		IF PULSO_CNT_L4_1T.Q = FALSE AND PULSO_CNT_L4_2T.Q = FALSE AND PULSO_CNT_L4_3T.Q = FALSE  THEN
		HabTemParadaL4 := TRUE;
		
		ELSE 	
		HabTemParadaL4 := FALSE;
		END_IF
		//LÓGICA PARA CONTAR TEMPO DE PARADA
//==============Habilita contadores 1º turno ================
IF (hora = HoraInicio1Turno AND minuto = MinInicio1Turno)  THEN
HabContL4_1T := TRUE;
HabContL4_3T := FALSE;
HabContL4_2T := FALSE;
CNT_PRD_L4_3T := 0;
CNT_PRD_L4_2T := 0;
CNT_PRD_L4_1T := 0;
TempoProduzindoL4 :=0;
EficL4_1T_projetada:=0;
EficL4_1T_realtime :=0;
ProdL4_1T_realtime :=0;
TempoParadaL4 :=0;
CXS_ATRASOL4:=0;
END_IF 


//==============Contador e Eficiencia L4 1 TURNO de cartuchos==========
IF HabContL4_1T = TRUE THEN 
PULSO_CNT_L4_1T(CLK:=CNT_L4);
//TMR_SIMUL_CNT1(IN:=LIBERA_TMR_SIMUL ,PT:=T#9S);	
		IF PULSO_CNT_L4_1T.Q = TRUE THEN
		CNT_PRD_L4_1T := CNT_PRD_L4_1T+1;
		//LIBERA_TMR_SIMUL := FALSE;
		RegistraHora := FALSE;
		MinDispTurnoAtual := MinDispL4_1T;
//ELSE 	
	//LIBERA_TMR_SIMUL:= TRUE;
		END_IF
		
			IF hora > 5 AND hora < 11 THEN

		ProdL4_1T_realtime := (INT_TO_REAL(ProducaoProgramada_L4_1T) / (MinDispL4_1T)) * ((
		(INT_TO_REAL(hora)-INT_TO_REAL(HoraInicio1Turno))*60)-INT_TO_REAL(MinInicio1Turno) + INT_TO_REAL(minuto));
		
		TempoProduzindoL4 :=  ((hora-HoraInicio1Turno)*60)-MinInicio1Turno+ minuto-TempoParadaL4;
		
		EficL4_1T_realtime := ( INT_TO_REAL(CNT_PRD_L4_1T) / ProdL4_1T_realtime ) * 100 * (EficL4_1T_projetada/100);
		EficL4_1T_projetada := (ProdL4_1T_realtime / ProducaoProgramada_L4_1T) * 100;
		END_IF
		
			IF hora > 11 AND hora < 15 THEN

		ProdL4_1T_realtime := (INT_TO_REAL(ProducaoProgramada_L4_1T) / (MinDispL4_1T)) * ((
		(INT_TO_REAL(hora)-INT_TO_REAL(HoraInicio1Turno))*60)-INT_TO_REAL(MinInicio1Turno) + INT_TO_REAL(minuto)-10-60);
		
		TempoProduzindoL4 :=  ((hora-HoraInicio1Turno)*60)-MinInicio1Turno+ minuto-TempoParadaL4;
		
		EficL4_1T_realtime := ( INT_TO_REAL(CNT_PRD_L4_1T) / ProdL4_1T_realtime ) * 100 * (EficL4_1T_projetada/100);
		EficL4_1T_projetada := (ProdL4_1T_realtime / ProducaoProgramada_L4_1T) * 100;
		END_IF
	
END_IF
EficienciaL4_1T := (INT_TO_REAL(CNT_PRD_L4_1T) / INT_TO_REAL(ProducaoProgramada_L4_1T) ) * 100;


//=====================1º TURNO ========================

//=====================2º TURNO ========================

	//10 minutos - Reunião / DSS / Treinamento
	//20 minutosPartida de linha / Parada de Linha
	//15 minutosRefeições (Café / Almoço / Janta)
	//60 minutosRefeições (Café / Almoço / Janta)
	//10 minutosPartida de linha / Parada de Linha
	IF hora = 0 THEN 
		hora := 24;
	END_IF
	
		MinDispL4_2T := (((INT_TO_REAL (HoraFim2Turno) - INT_TO_REAL(HoraInicio2Turno) )*60)-
		INT_TO_REAL(MinInicio2Turno)+INT_TO_REAL(MinFim2Turno)-60-10);
	
//==============Contador e Eficiencia L4 2 TURNO de cartuchos==========
//==============Habilita contadores 2º turno ================
IF (hora = HoraInicio2Turno AND minuto = MinInicio2Turno)  THEN
HabContL4_2T := TRUE;
HabContL4_1T := FALSE;
CNT_PRD_L4_3T := 0;
CNT_PRD_L4_2T := 0;
CNT_PRD_L4_1T := 0;
TempoParadaL4 :=0;
TempoProduzindoL4 :=0;
EficL4_1T_projetada:=0;
EficL4_1T_realtime :=0;
ProdL4_1T_realtime :=0;
TempoParadaL4 :=0;
CXS_ATRASOL4:=0;
END_IF 
IF HabContL4_2T = TRUE THEN 
PULSO_CNT_L4_2T(CLK:=CNT_L4);
//TMR_SIMUL_CNT2(IN:=LIBERA_TMR_SIMUL4T ,PT:=T#7S);
		IF PULSO_CNT_L4_2T.Q = TRUE  THEN
		CNT_PRD_L4_2T := CNT_PRD_L4_2T+1;
		//LIBERA_TMR_SIMUL4T := FALSE;
		MinDispTurnoAtual := MinDispL4_2T;
//ELSE 	
	//LIBERA_TMR_SIMUL4T:= TRUE;	
		END_IF
		CNT_PRD_L4_1T := CNT_PRD_L4_2T ;
		EficL4_1T_projetada:=EficL4_2T_projetada;
		EficL4_1T_realtime :=EficL4_2T_realtime;
		ProdL4_1T_realtime :=ProdL4_1T_realtime;
		
			IF hora > 13 AND hora < 19 THEN

		ProdL4_2T_realtime := (INT_TO_REAL(ProducaoProgramada_L4_T2) / (MinDispL4_2T)) * ((
		(INT_TO_REAL(hora)-INT_TO_REAL(HoraInicio2Turno))*60)-INT_TO_REAL(MinInicio2Turno) + INT_TO_REAL(minuto));
		
		TempoProduzindoL4 :=  ((hora-HoraInicio2Turno)*60)-MinInicio2Turno+ minuto-TempoParadaL4;
		
		EficL4_2T_realtime := ( INT_TO_REAL(CNT_PRD_L4_2T) / ProdL4_2T_realtime ) * 100 * (EficL4_2T_projetada/100);
		EficL4_2T_projetada := (ProdL4_2T_realtime / ProducaoProgramada_L4_T2) * 100;
		END_IF
		IF hora > 19 AND hora < 23 THEN

		ProdL4_2T_realtime := (INT_TO_REAL(ProducaoProgramada_L4_T2) / (MinDispL4_2T)) * ((
		(INT_TO_REAL(hora)-INT_TO_REAL(HoraInicio2Turno))*60)-INT_TO_REAL(MinInicio2Turno) + INT_TO_REAL(minuto)-10-60);
		
		TempoProduzindoL4 :=  ((hora-HoraInicio2Turno)*60)-MinInicio2Turno+ minuto-TempoParadaL4;
		
		EficL4_2T_realtime := ( INT_TO_REAL(CNT_PRD_L4_2T) / ProdL4_2T_realtime ) * 100 * (EficL4_2T_projetada/100);
		EficL4_2T_projetada := (ProdL4_2T_realtime / ProducaoProgramada_L4_T2) * 100;
		END_IF
END_IF
EficienciaL4_2T := (INT_TO_REAL (CNT_PRD_L4_2T) / INT_TO_REAL (ProducaoProgramada_L4_T2)  ) * 100;

//=====================2º TURNO ========================

//=====================3º TURNO ========================
//==============Contador e Eficiencia L4 3 TURNO de cartuchos==========

//==============Habilita contadores 3º turno ================
//10 minutos - Reunião / DSS / Treinamento
	//20 minutosPartida de linha / Parada de Linha
	//15 minutosRefeições (Café / Almoço / Janta)
	//60 minutosRefeições (Café / Almoço / Janta)
	//10 minutosPartida de linha / Parada de Linha
	IF hora = 0 THEN 
		hora := 24;
	END_IF
	
		MinDispL4_3T := (((INT_TO_REAL (HoraFim3Turno) - INT_TO_REAL(HoraInicio3Turno) )*60)-
		INT_TO_REAL(MinInicio3Turno)+INT_TO_REAL(MinFim3Turno)-60-10);
		
	
//==============Contador e Eficiencia L4 3 TURNO de cartuchos==========
//==============Habilita contadores 3º turno ================
IF (hora = HoraInicio3Turno AND minuto = MinInicio3Turno)  THEN
HabContL4_3T := TRUE;
HabContL4_2T := FALSE;
HabContL4_1T := FALSE;
CNT_PRD_L4_3T := 0;
CNT_PRD_L4_2T := 0;
CNT_PRD_L4_1T := 0;
TempoParadaL4 :=0;
TempoProduzindoL4 :=0;
EficL4_1T_projetada:=0;
EficL4_1T_realtime :=0;
ProdL4_1T_realtime :=0;
TempoParadaL4 :=0;
CXS_ATRASOL4:=0;
END_IF 

IF HabContL4_3T = TRUE THEN 
PULSO_CNT_L4_3T(CLK:=CNT_L4);	
		IF PULSO_CNT_L4_3T.Q = TRUE THEN
		CNT_PRD_L4_3T := CNT_PRD_L4_3T+1;	
			CNT_PRD_L4_1T := CNT_PRD_L4_3T ;
		EficL4_1T_projetada:=EficL4_3T_projetada;
		EficL4_1T_realtime :=EficL4_3T_realtime;
		ProdL4_1T_realtime :=ProdL4_3T_realtime;
		END_IF
		IF hora > 21 AND hora <= 24 THEN

		ProdL4_3T_realtime := (INT_TO_REAL(ProducaoProgramada_L4_T3) / (MinDispL4_3T)) * ((
		(INT_TO_REAL(hora)-INT_TO_REAL(HoraInicio3Turno))*60)-INT_TO_REAL(MinInicio3Turno) + INT_TO_REAL(minuto));
		
		TempoProduzindoL4 :=  ((hora-HoraInicio3Turno)*60)-MinInicio3Turno+ minuto-TempoParadaL4;
	
		EficL4_3T_realtime := ( INT_TO_REAL(CNT_PRD_L4_3T) / ProdL4_3T_realtime ) * 100 *(EficL4_3T_projetada/100) ;
		EficL4_3T_projetada := (ProdL4_3T_realtime / ProducaoProgramada_L4_T3) * 100;
		END_IF
		IF ((hora > 0 ) AND minuto > 30) AND hora < 2 THEN

		ProdL4_3T_realtime := (INT_TO_REAL(ProducaoProgramada_L4_T3) / (MinDispL4_3T)) * ((
		(INT_TO_REAL(hora)-INT_TO_REAL(HoraInicio3Turno))*60)-INT_TO_REAL(MinInicio3Turno) + INT_TO_REAL(minuto)-10-60);
		
		TempoProduzindoL4 :=  ((hora-HoraInicio3Turno)*60)-MinInicio3Turno+ minuto-TempoParadaL4;
	
		EficL4_3T_realtime := ( INT_TO_REAL(CNT_PRD_L4_3T) / ProdL4_3T_realtime ) * 100 *(EficL4_3T_projetada/100) ;
		EficL4_3T_projetada := (ProdL4_3T_realtime / ProducaoProgramada_L4_T3) * 100;
		END_IF
END_IF


EficienciaL4_3T := (INT_TO_REAL (CNT_PRD_L4_3T) / INT_TO_REAL (ProducaoProgramada_L4_T3)  ) * 100;


IF (hora = HoraInicio3Turno AND minuto = MinInicio3Turno)  THEN
HabContL4_3T := TRUE;
HabContL4_2T := FALSE;
END_IF 

IF HabContL4_3T = TRUE THEN 
PULSO_CNT_L4_3T(CLK:=CNT_L4);
//TMR_SIMUL_CNT3(IN:=LIBERA_TMR_SIMUL4T ,PT:=T#8S);
		IF PULSO_CNT_L4_3T.Q = TRUE  THEN
		CNT_PRD_L4_3T := CNT_PRD_L4_3T+1;
		//LIBERA_TMR_SIMUL4T := FALSE;
		MinDispTurnoAtual := MinDispL4_3T;
//ELSE 	
	//LIBERA_TMR_SIMUL4T:= TRUE;	
		END_IF
		END_IF
	
	
EficienciaL4_3T := (INT_TO_REAL (CNT_PRD_L4_3T) / INT_TO_REAL(ProducaoProgramada_L4_T3)  ) * 100;
//=====================3º TURNO ========================

IF (hora = 11 AND minuto = 0) OR (hora = 19 AND minuto = 0) OR (hora = 1 AND minuto = 30)  THEN
	refeicao := TRUE;
	END_IF
	IF (hora = 11 AND minuto = 40) OR  (hora = 20 AND minuto = 0)  OR  (hora = 2 AND minuto = 30)  THEN
	refeicao := FALSE;
	END_IF 
	
	IF (hora = 6 AND minuto = 0) OR (hora = 20 AND minuto = 0) OR (hora = 2 AND minuto = 30)  THEN
	DDS := TRUE;
	END_IF
	IF (hora = 6 AND minuto = 10) OR  (hora = 20 AND minuto = 10)  OR  (hora = 2 AND minuto = 40)  THEN
	DDS := FALSE;
	END_IF 
	IF (hora = 6 AND minuto = 0) OR (hora = 14 AND minuto = 20) OR (hora = 22 AND minuto = 30)  THEN
	SETUP := TRUE;
	END_IF
	IF (hora = 6 AND minuto = 30) OR  (hora = 14 AND minuto = 50)  OR  (hora = 23 AND minuto = 0)  THEN
	SETUP := FALSE;
	END_IF 
	
	
//STATUS DA LINHA 4
//STATUS DO EQUIPAMENTO
//0- SEM PROGRAMAÇÃO
//1- PRODUZINDO
//2- PARADA
//3- REFEIÇÃO
//4- DDS
//5- SETUP

	
IF ProducaoProgramada_L4_1T = 0 AND HabContL4_1T  AND TempParadaL4.Q = TRUE THEN
	Status_L4 := 0;
	L4semprogramacao :=TRUE;
	END_IF
		IF ProducaoProgramada_L4_1T > 0 AND HabContL4_1T = TRUE THEN 
		L4semprogramacao :=FALSE;
		END_IF
	
IF ProducaoProgramada_L4_T2 = 0 AND HabContL4_2T = TRUE AND TempParadaL4.Q = TRUE THEN
	Status_L4 := 0;
	L4semprogramacao :=TRUE;
		END_IF
			IF ProducaoProgramada_L4_T2 > 0 AND HabContL4_2T = TRUE THEN 
				L4semprogramacao :=FALSE;
				END_IF
				
IF ProducaoProgramada_L4_T3 = 0 AND HabContL4_3T = TRUE AND TempParadaL4.Q = TRUE THEN
	Status_L4 := 0;
	L4semprogramacao :=TRUE;
		END_IF
			IF ProducaoProgramada_L4_T3 > 0 AND HabContL4_3T = TRUE THEN 
			L4semprogramacao :=FALSE;
			END_IF
	
IF  TempParadaL4.Q = FALSE  THEN
	Status_L4 := 1;
END_IF

	IF refeicao = FALSE AND SETUP = FALSE AND DDS = FALSE AND TempParadaL4.Q = TRUE AND L4semprogramacao = FALSE THEN
	Status_L4 := 2;
	END_IF

IF refeicao = TRUE AND TempParadaL4.Q = TRUE  THEN
Status_L4 := 3;
END_IF

IF DDS = TRUE AND TempParadaL4.Q = TRUE THEN
Status_L4 := 4;
END_IF

//IF SETUP = TRUE THEN
//Status_L4 := 5;
//END_IF
//STATUS DA LINHA 4

END_PROGRAM

// Device/Application/ProdL5
PROGRAM ProdL5
VAR
	//PRODUÇÃO LINHAS ENVASE
	
//=========================	
PULSO_CNT_L5_1T: R_TRIG;
PULSO_CNT_L5_2T: R_TRIG;
PULSO_CNT_L5_3T: R_TRIG;
	CNT_PRD_L5: INT;
	//CNT_L5: BOOL;
//=========================	
	Result : RTC_STATUS;
	DATEANDTIME : EXTENDED_DATE_AND_TIME;
	xEnable : BOOL;
//=========================		
	dia: INT;
	mes: INT;
	ano: INT;
	hora: INT;
	minuto: INT;
	segundo: INT;
	
	
	
	//HoraInicio1Turno: INT;
	//MinInicio1Turno: INT;
	HoraFim1Turno: INT;
	MinFim1Turno: INT;
	//HoraInicio2Turno: INT;
	//MinInicio2Turno: INT;
	HoraFim2Turno: INT;
	MinFim2Turno: INT;
	//HoraInicio3Turno: INT;
	//MinInicio3Turno: INT;
	HoraFim3Turno: INT;
	MinFim3Turno: INT;
	EficienciaL5: INT;
	
	
	HabContL5_1T: BOOL;
	HabContL5_2T: BOOL;
	HabContL5_3T: BOOL;
	
	CNT_PRD_L5_2T: INT;
	CNT_PRD_L5_3T: INT;
	EficienciaL5_1T: REAL;
	EficienciaL5_2T: REAL;
	EficienciaL5_3T: REAL;
	
	MinDispL5_1T: REAL;
	
	ProdL5_1T_realtime: REAL;
	MinDispL5_2T: REAL;
	ProdL5_2T_realtime: REAL;
	EficL5_2T_realtime: REAL;
	MinDispL5_3T: REAL;
	ProdL5_3T_realtime: REAL;
	EficL5_3T_realtime: REAL;
	
	//TMR_SIMUL_CNT1: TON;
	//LIBERA_TMR_SIMUL: BOOL;
	EficL5_2T_projetada: REAL;
	//TMR_SIMUL_CNT2: TON;
	//LIBERA_TMR_SIMUL5T: BOOL;
	//TMR_SIMUL_CNT3: TON;
	//LIBERA_TMR_SIMUL5T: BOOL;
	EficL5_3T_projetada: REAL;
//	EficL5_1T_realtime: REAL;
	HabTemParadaL5: BOOL;
	TempParadaL5: Ton;
	horaParadaL5: INT;
	MinParadaL5: INT;
	RegistraHora: BOOL;
	Borda_des_RegistraHora: F_TRIG;
	HoraRetornoParadaL5: INT;
	MinRetornoParadaL5: INT;
	TempoParadaL5L5: INT;
	TotalMinParado: TON;
	HabTotalMinParado: BOOL;
	//TempoProduzindoL5: REAL;
	//MinDispTurnoAtual: REAL;

	refeicao: BOOL;
	DDS: BOOL;
	SETUP: BOOL;
	L5semprogramacao: BOOL;
END_VAR


//LÓGICA PARA ANÁLISES DE PRODUTIVADADE DA L5 DE CARTUCHOS
	dia := BYTE_TO_INT (DATEANDTIME.byDayOfMonth);
	mes := BYTE_TO_INT (DATEANDTIME.byMonth);
	ano := WORD_TO_INT (DATEANDTIME.wYear);
	hora := BYTE_TO_INT (DATEANDTIME.byHours);
	minuto := BYTE_TO_INT (DATEANDTIME.byMinutes);
	segundo := BYTE_TO_INT (DATEANDTIME.bySeconds);
	xEnable := TRUE;
	
	//HABILITA RTC==========================
	IF xEnable = TRUE THEN
	Result := GetDateAndTime(DATEANDTIME);
	END_IF
//HABILITA RTC==========================

//=====================1º TURNO ========================
	
		//HoraInicio1Turno: INT;
	
	HoraFim1Turno:= HoraInicio2Turno;
	MinFim1Turno:= MinInicio2Turno;
	HoraFim2Turno:= HoraInicio3Turno;
	MinFim2Turno:= MinInicio3Turno;
	
	//10 minutos - Reunião / DSS / Treinamento
	//20 minutosPartida de linha / Parada de Linha xxxxxxxxxx
	//15 minutosRefeições (Café / Almoço / Janta)xxxxxxxxxxxx
	//60 minutosRefeições (Café / Almoço / Janta)
	//10 minutosPartida de linha / Parada de Linha xxxxxxxxxxxxxx
			
	MinDispL5_1T := (((INT_TO_REAL (HoraFim1Turno) - INT_TO_REAL(HoraInicio1Turno) )*60)-
		INT_TO_REAL(MinInicio1Turno)+INT_TO_REAL(MinFim1Turno)-60-10);
		
			IF TempoProduzindoL5 < 1 THEN
			TempoProduzindoL5 :=0;
		END_IF
	
			//LÓGICA PARA VERIFICAR SE EXISTE ATRASO DE PRODUÇÃO NO INSTANTE ATUAL
		
	IF  CXS_ATRASOL5 >= 0 AND HabContL5_1T = TRUE THEN 
	CXS_ATRASOL5:= REAL_TO_INT(ProdL5_1T_realtime)-CNT_PRD_L5_1T;
	END_IF
	IF  CXS_ATRASOL5 >= 0 AND HabContL5_2T = TRUE THEN 
	CXS_ATRASOL5:= REAL_TO_INT(ProdL5_2T_realtime)-CNT_PRD_L5_1T;
	END_IF
	IF  CXS_ATRASOL5 >= 0 AND HabContL5_3T = TRUE THEN 
	CXS_ATRASOL5:=REAL_TO_INT(ProdL5_2T_realtime)-CNT_PRD_L5_1T;
	END_IF
		IF  CXS_ATRASOL5  < 0 THEN 
		CXS_ATRASOL5:= 0;
		END_IF
	
	
	//LÓGICA PARA VERIFICAR SE EXISTE ATRASO DE PRODUÇÃO NO INSTANTE ATUAL
	
		
		//LÓGICA PARA CONTAR TEMPO DE PARADA
		TempParadaL5(IN:=HabTemParadaL5 ,PT:= T#30S);
		IF TempParadaL5.Q   THEN
		TotalMinParado(IN:=HabTotalMinParado ,PT:= T#1M);
		IF TotalMinParado.Q = TRUE THEN
			TempoParadaL5 := TempoParadaL5+1;
			HabTotalMinParado := FALSE;
			ELSE
				HabTotalMinParado := TRUE;
			END_IF
		END_IF
		
		IF PULSO_CNT_L5_1T.Q = FALSE AND PULSO_CNT_L5_2T.Q = FALSE AND PULSO_CNT_L5_3T.Q = FALSE  THEN
		HabTemParadaL5 := TRUE;
		
		ELSE 	
		HabTemParadaL5 := FALSE;
		END_IF
		//LÓGICA PARA CONTAR TEMPO DE PARADA
//==============Habilita contadores 1º turno ================
IF (hora = HoraInicio1Turno AND minuto = MinInicio1Turno)  THEN
HabContL5_1T := TRUE;
HabContL5_3T := FALSE;
HabContL5_2T := FALSE;
CNT_PRD_L5_3T := 0;
CNT_PRD_L5_2T := 0;
CNT_PRD_L5_1T := 0;
TempoProduzindoL5 :=0;
EficL5_1T_projetada:=0;
EficL5_1T_realtime :=0;
ProdL5_1T_realtime :=0;
TempoParadaL5 :=0;
CXS_ATRASOL5:=0;
END_IF 


//==============Contador e Eficiencia L5 1 TURNO de cartuchos==========
IF HabContL5_1T = TRUE THEN 
PULSO_CNT_L5_1T(CLK:=CNT_L5);
//TMR_SIMUL_CNT1(IN:=LIBERA_TMR_SIMUL ,PT:=T#9S);	
		IF PULSO_CNT_L5_1T.Q = TRUE THEN
		CNT_PRD_L5_1T := CNT_PRD_L5_1T+1;
		//LIBERA_TMR_SIMUL := FALSE;
		RegistraHora := FALSE;
		MinDispTurnoAtual := MinDispL5_1T;
//ELSE 	
	//LIBERA_TMR_SIMUL:= TRUE;
		END_IF
		
			IF hora > 5 AND hora < 11 THEN

		ProdL5_1T_realtime := (INT_TO_REAL(ProducaoProgramada_L5_1T) / (MinDispL5_1T)) * ((
		(INT_TO_REAL(hora)-INT_TO_REAL(HoraInicio1Turno))*60)-INT_TO_REAL(MinInicio1Turno) + INT_TO_REAL(minuto));
		
		TempoProduzindoL5 :=  ((hora-HoraInicio1Turno)*60)-MinInicio1Turno+ minuto-TempoParadaL5;
		
		EficL5_1T_realtime := ( INT_TO_REAL(CNT_PRD_L5_1T) / ProdL5_1T_realtime ) * 100 * (EficL5_1T_projetada/100);
		EficL5_1T_projetada := (ProdL5_1T_realtime / ProducaoProgramada_L5_1T) * 100;
		END_IF
		
			IF hora > 11 AND hora < 15 THEN

		ProdL5_1T_realtime := (INT_TO_REAL(ProducaoProgramada_L5_1T) / (MinDispL5_1T)) * ((
		(INT_TO_REAL(hora)-INT_TO_REAL(HoraInicio1Turno))*60)-INT_TO_REAL(MinInicio1Turno) + INT_TO_REAL(minuto)-10-60);
		
		TempoProduzindoL5 :=  ((hora-HoraInicio1Turno)*60)-MinInicio1Turno+ minuto-TempoParadaL5;
		
		EficL5_1T_realtime := ( INT_TO_REAL(CNT_PRD_L5_1T) / ProdL5_1T_realtime ) * 100 * (EficL5_1T_projetada/100);
		EficL5_1T_projetada := (ProdL5_1T_realtime / ProducaoProgramada_L5_1T) * 100;
		END_IF
	
END_IF
EficienciaL5_1T := (INT_TO_REAL(CNT_PRD_L5_1T) / INT_TO_REAL(ProducaoProgramada_L5_1T) ) * 100;


//=====================1º TURNO ========================

//=====================2º TURNO ========================

	//10 minutos - Reunião / DSS / Treinamento
	//20 minutosPartida de linha / Parada de Linha
	//15 minutosRefeições (Café / Almoço / Janta)
	//60 minutosRefeições (Café / Almoço / Janta)
	//10 minutosPartida de linha / Parada de Linha
	IF hora = 0 THEN 
		hora := 24;
	END_IF
	
		MinDispL5_2T := (((INT_TO_REAL (HoraFim2Turno) - INT_TO_REAL(HoraInicio2Turno) )*60)-
		INT_TO_REAL(MinInicio2Turno)+INT_TO_REAL(MinFim2Turno)-60-10);
	
//==============Contador e Eficiencia L5 2 TURNO de cartuchos==========
//==============Habilita contadores 2º turno ================
IF (hora = HoraInicio2Turno AND minuto = MinInicio2Turno)  THEN
HabContL5_2T := TRUE;
HabContL5_1T := FALSE;
CNT_PRD_L5_3T := 0;
CNT_PRD_L5_2T := 0;
CNT_PRD_L5_1T := 0;
TempoParadaL5 :=0;
TempoProduzindoL5 :=0;
EficL5_1T_projetada:=0;
EficL5_1T_realtime :=0;
ProdL5_1T_realtime :=0;
TempoParadaL5 :=0;
CXS_ATRASOL5:=0;
END_IF 
IF HabContL5_2T = TRUE THEN 
PULSO_CNT_L5_2T(CLK:=CNT_L5);
//TMR_SIMUL_CNT2(IN:=LIBERA_TMR_SIMUL5T ,PT:=T#7S);
		IF PULSO_CNT_L5_2T.Q = TRUE  THEN
		CNT_PRD_L5_2T := CNT_PRD_L5_2T+1;
		//LIBERA_TMR_SIMUL5T := FALSE;
		MinDispTurnoAtual := MinDispL5_2T;
//ELSE 	
	//LIBERA_TMR_SIMUL5T:= TRUE;	
		END_IF
		CNT_PRD_L5_1T := CNT_PRD_L5_2T ;
		EficL5_1T_projetada:=EficL5_2T_projetada;
		EficL5_1T_realtime :=EficL5_2T_realtime;
		ProdL5_1T_realtime :=ProdL5_1T_realtime;
		
			IF hora > 13 AND hora < 19 THEN

		ProdL5_2T_realtime := (INT_TO_REAL(ProducaoProgramada_L5_T2) / (MinDispL5_2T)) * ((
		(INT_TO_REAL(hora)-INT_TO_REAL(HoraInicio2Turno))*60)-INT_TO_REAL(MinInicio2Turno) + INT_TO_REAL(minuto));
		
		TempoProduzindoL5 :=  ((hora-HoraInicio2Turno)*60)-MinInicio2Turno+ minuto-TempoParadaL5;
		
		EficL5_2T_realtime := ( INT_TO_REAL(CNT_PRD_L5_2T) / ProdL5_2T_realtime ) * 100 * (EficL5_2T_projetada/100);
		EficL5_2T_projetada := (ProdL5_2T_realtime / ProducaoProgramada_L5_T2) * 100;
		END_IF
		IF hora > 19 AND hora < 23 THEN

		ProdL5_2T_realtime := (INT_TO_REAL(ProducaoProgramada_L5_T2) / (MinDispL5_2T)) * ((
		(INT_TO_REAL(hora)-INT_TO_REAL(HoraInicio2Turno))*60)-INT_TO_REAL(MinInicio2Turno) + INT_TO_REAL(minuto)-10-60);
		
		TempoProduzindoL5 :=  ((hora-HoraInicio2Turno)*60)-MinInicio2Turno+ minuto-TempoParadaL5;
		
		EficL5_2T_realtime := ( INT_TO_REAL(CNT_PRD_L5_2T) / ProdL5_2T_realtime ) * 100 * (EficL5_2T_projetada/100);
		EficL5_2T_projetada := (ProdL5_2T_realtime / ProducaoProgramada_L5_T2) * 100;
		END_IF
END_IF
EficienciaL5_2T := (INT_TO_REAL (CNT_PRD_L5_2T) / INT_TO_REAL (ProducaoProgramada_L5_T2)  ) * 100;

//=====================2º TURNO ========================

//=====================3º TURNO ========================
//==============Contador e Eficiencia L5 3 TURNO de cartuchos==========

//==============Habilita contadores 3º turno ================
//10 minutos - Reunião / DSS / Treinamento
	//20 minutosPartida de linha / Parada de Linha
	//15 minutosRefeições (Café / Almoço / Janta)
	//60 minutosRefeições (Café / Almoço / Janta)
	//10 minutosPartida de linha / Parada de Linha
	IF hora = 0 THEN 
		hora := 24;
	END_IF
	
		MinDispL5_3T := (((INT_TO_REAL (HoraFim3Turno) - INT_TO_REAL(HoraInicio3Turno) )*60)-
		INT_TO_REAL(MinInicio3Turno)+INT_TO_REAL(MinFim3Turno)-60-10);
		
	
//==============Contador e Eficiencia L5 3 TURNO de cartuchos==========
//==============Habilita contadores 3º turno ================
IF (hora = HoraInicio3Turno AND minuto = MinInicio3Turno)  THEN
HabContL5_3T := TRUE;
HabContL5_2T := FALSE;
HabContL5_1T := FALSE;
CNT_PRD_L5_3T := 0;
CNT_PRD_L5_2T := 0;
CNT_PRD_L5_1T := 0;
TempoParadaL5 :=0;
TempoProduzindoL5 :=0;
EficL5_1T_projetada:=0;
EficL5_1T_realtime :=0;
ProdL5_1T_realtime :=0;
TempoParadaL5 :=0;
CXS_ATRASOL5:=0;
END_IF 

IF HabContL5_3T = TRUE THEN 
PULSO_CNT_L5_3T(CLK:=CNT_L5);	
		IF PULSO_CNT_L5_3T.Q = TRUE THEN
		CNT_PRD_L5_3T := CNT_PRD_L5_3T+1;	
			CNT_PRD_L5_1T := CNT_PRD_L5_3T ;
		EficL5_1T_projetada:=EficL5_3T_projetada;
		EficL5_1T_realtime :=EficL5_3T_realtime;
		ProdL5_1T_realtime :=ProdL5_3T_realtime;
		END_IF
		IF hora > 21 AND hora <= 24 THEN

		ProdL5_3T_realtime := (INT_TO_REAL(ProducaoProgramada_L5_T3) / (MinDispL5_3T)) * ((
		(INT_TO_REAL(hora)-INT_TO_REAL(HoraInicio3Turno))*60)-INT_TO_REAL(MinInicio3Turno) + INT_TO_REAL(minuto));
		
		TempoProduzindoL5 :=  ((hora-HoraInicio3Turno)*60)-MinInicio3Turno+ minuto-TempoParadaL5;
	
		EficL5_3T_realtime := ( INT_TO_REAL(CNT_PRD_L5_3T) / ProdL5_3T_realtime ) * 100 *(EficL5_3T_projetada/100) ;
		EficL5_3T_projetada := (ProdL5_3T_realtime / ProducaoProgramada_L5_T3) * 100;
		END_IF
		IF ((hora > 0 ) AND minuto > 30) AND hora < 2 THEN

		ProdL5_3T_realtime := (INT_TO_REAL(ProducaoProgramada_L5_T3) / (MinDispL5_3T)) * ((
		(INT_TO_REAL(hora)-INT_TO_REAL(HoraInicio3Turno))*60)-INT_TO_REAL(MinInicio3Turno) + INT_TO_REAL(minuto)-10-60);
		
		TempoProduzindoL5 :=  ((hora-HoraInicio3Turno)*60)-MinInicio3Turno+ minuto-TempoParadaL5;
	
		EficL5_3T_realtime := ( INT_TO_REAL(CNT_PRD_L5_3T) / ProdL5_3T_realtime ) * 100 *(EficL5_3T_projetada/100) ;
		EficL5_3T_projetada := (ProdL5_3T_realtime / ProducaoProgramada_L5_T3) * 100;
		END_IF
END_IF


EficienciaL5_3T := (INT_TO_REAL (CNT_PRD_L5_3T) / INT_TO_REAL (ProducaoProgramada_L5_T3)  ) * 100;


IF (hora = HoraInicio3Turno AND minuto = MinInicio3Turno)  THEN
HabContL5_3T := TRUE;
HabContL5_2T := FALSE;
END_IF 

IF HabContL5_3T = TRUE THEN 
PULSO_CNT_L5_3T(CLK:=CNT_L5);
//TMR_SIMUL_CNT3(IN:=LIBERA_TMR_SIMUL5T ,PT:=T#8S);
		IF PULSO_CNT_L5_3T.Q = TRUE  THEN
		CNT_PRD_L5_3T := CNT_PRD_L5_3T+1;
		//LIBERA_TMR_SIMUL5T := FALSE;
		MinDispTurnoAtual := MinDispL5_3T;
//ELSE 	
	//LIBERA_TMR_SIMUL5T:= TRUE;	
		END_IF
		END_IF
	
	
EficienciaL5_3T := (INT_TO_REAL (CNT_PRD_L5_3T) / INT_TO_REAL(ProducaoProgramada_L5_T3)  ) * 100;
//=====================3º TURNO ========================

IF (hora = 11 AND minuto = 0) OR (hora = 19 AND minuto = 0) OR (hora = 1 AND minuto = 30)  THEN
	refeicao := TRUE;
	END_IF
	IF (hora = 11 AND minuto = 40) OR  (hora = 20 AND minuto = 0)  OR  (hora = 2 AND minuto = 30)  THEN
	refeicao := FALSE;
	END_IF 
	
	IF (hora = 6 AND minuto = 0) OR (hora = 20 AND minuto = 0) OR (hora = 2 AND minuto = 30)  THEN
	DDS := TRUE;
	END_IF
	IF (hora = 6 AND minuto = 10) OR  (hora = 20 AND minuto = 10)  OR  (hora = 2 AND minuto = 40)  THEN
	DDS := FALSE;
	END_IF 
	IF (hora = 6 AND minuto = 0) OR (hora = 14 AND minuto = 20) OR (hora = 22 AND minuto = 30)  THEN
	SETUP := TRUE;
	END_IF
	IF (hora = 6 AND minuto = 30) OR  (hora = 14 AND minuto = 50)  OR  (hora = 23 AND minuto = 0)  THEN
	SETUP := FALSE;
	END_IF 
	
//STATUS DA LINHA =5
//STATUS DO EQUIPAMENTO
//0- SEM PROGRAMAÇÃO
//1- PRODUZINDO
//2- PARADA
//3- REFEIÇÃO
//4- DDS
//5- SETUP

IF ProducaoProgramada_L5_1T = 0 AND HabContL5_1T = TRUE AND TempParadaL5.Q = TRUE THEN
	Status_L5 := 0;
	L5semprogramacao :=TRUE;
	END_IF
		IF ProducaoProgramada_L5_1T > 0 AND HabContL5_1T = TRUE THEN 
		L5semprogramacao :=FALSE;
		END_IF
	
IF ProducaoProgramada_L5_T2 = 0 AND HabContL5_2T = TRUE AND TempParadaL5.Q = TRUE THEN
	Status_L5 := 0;
	L5semprogramacao :=TRUE;
		END_IF
			IF ProducaoProgramada_L5_T2 > 0 AND HabContL5_2T = TRUE THEN 
				L5semprogramacao :=FALSE;
				END_IF
				
IF ProducaoProgramada_L5_T3 = 0 AND HabContL5_3T = TRUE AND TempParadaL5.Q = TRUE THEN
	Status_L5 := 0;
	L5semprogramacao :=TRUE;
		END_IF
			IF ProducaoProgramada_L5_T3 > 0 AND HabContL5_3T = TRUE THEN 
			L5semprogramacao :=FALSE;
			END_IF
	
IF  TempParadaL5.Q = FALSE  THEN
	Status_L5 := 1;
END_IF

	IF refeicao = FALSE AND SETUP = FALSE AND DDS = FALSE AND TempParadaL5.Q = TRUE AND L5semprogramacao = FALSE THEN
	Status_L5 := 2;
	END_IF

IF refeicao = TRUE  AND TempParadaL5.Q = TRUE THEN
Status_L5 := 3;
END_IF

IF DDS = TRUE  AND TempParadaL5.Q = TRUE THEN
Status_L5 := 4;
END_IF

//IF SETUP = TRUE THEN
//Status_L5 := 5;
//END_IF
//STATUS DA LINHA 5

END_PROGRAM

// Device/Application/ProdL6
PROGRAM ProdL6
VAR
	//PRODUÇÃO LINHAS ENVASE
	
//=========================	
PULSO_CNT_L6_1T: R_TRIG;
PULSO_CNT_L6_2T: R_TRIG;
PULSO_CNT_L6_3T: R_TRIG;
	CNT_PRD_L6: INT;
	//CNT_L6: BOOL;
//=========================	
	Result : RTC_STATUS;
	DATEANDTIME : EXTENDED_DATE_AND_TIME;
	xEnable : BOOL;
//=========================		
	dia: INT;
	mes: INT;
	ano: INT;
	hora: INT;
	minuto: INT;
	segundo: INT;
	
	
	
	//HoraInicio1Turno: INT;
	//MinInicio1Turno: INT;
	HoraFim1Turno: INT;
	MinFim1Turno: INT;
	//HoraInicio2Turno: INT;
	//MinInicio2Turno: INT;
	HoraFim2Turno: INT;
	MinFim2Turno: INT;
	//HoraInicio3Turno: INT;
	//MinInicio3Turno: INT;
	HoraFim3Turno: INT;
	MinFim3Turno: INT;
	EficienciaL6: INT;
	
	
	HabContL6_1T: BOOL;
	HabContL6_2T: BOOL;
	HabContL6_3T: BOOL;
	
	CNT_PRD_L6_2T: INT;
	CNT_PRD_L6_3T: INT;
	EficienciaL6_1T: REAL;
	EficienciaL6_2T: REAL;
	EficienciaL6_3T: REAL;
	
	MinDispL6_1T: REAL;
	
	ProdL6_1T_realtime: REAL;
	MinDispL6_2T: REAL;
	ProdL6_2T_realtime: REAL;
	EficL6_2T_realtime: REAL;
	MinDispL6_3T: REAL;
	ProdL6_3T_realtime: REAL;
	EficL6_3T_realtime: REAL;
	
	//TMR_SIMUL_CNT1: TON;
	//LIBERA_TMR_SIMUL: BOOL;
	EficL6_2T_projetada: REAL;
	//TMR_SIMUL_CNT2: TON;
	//LIBERA_TMR_SIMUL6T: BOOL;
	//TMR_SIMUL_CNT3: TON;
	//LIBERA_TMR_SIMUL3T: BOOL;
	EficL6_3T_projetada: REAL;
//	EficL6_1T_realtime: REAL;
	HabTemParadaL6: BOOL;
	TempParadaL6: Ton;
	horaParadaL6: INT;
	MinParadaL6: INT;
	RegistraHora: BOOL;
	Borda_des_RegistraHora: F_TRIG;
	HoraRetornoParadaL6: INT;
	MinRetornoParadaL6: INT;
	TempoParadaL6L6: INT;
	TotalMinParado: TON;
	HabTotalMinParado: BOOL;
	//TempoProduzindoL6: REAL;
	//MinDispTurnoAtual: REAL;

	refeicao: BOOL;
	DDS: BOOL;
	SETUP: BOOL;
	L6semprogramacao: BOOL;
END_VAR


//LÓGICA PARA ANÁLISES DE PRODUTIVADADE DA L6 DE CARTUCHOS
	dia := BYTE_TO_INT (DATEANDTIME.byDayOfMonth);
	mes := BYTE_TO_INT (DATEANDTIME.byMonth);
	ano := WORD_TO_INT (DATEANDTIME.wYear);
	hora := BYTE_TO_INT (DATEANDTIME.byHours);
	minuto := BYTE_TO_INT (DATEANDTIME.byMinutes);
	segundo := BYTE_TO_INT (DATEANDTIME.bySeconds);
	xEnable := TRUE;
	
	//HABILITA RTC==========================
	IF xEnable = TRUE THEN
	Result := GetDateAndTime(DATEANDTIME);
	END_IF
//HABILITA RTC==========================

//=====================1º TURNO ========================
	
		//HoraInicio1Turno: INT;
	
	HoraFim1Turno:= HoraInicio2Turno;
	MinFim1Turno:= MinInicio2Turno;
	HoraFim2Turno:= HoraInicio3Turno;
	MinFim2Turno:= MinInicio3Turno;
	
	//10 minutos - Reunião / DSS / Treinamento
	//20 minutosPartida de linha / Parada de Linha xxxxxxxxxx
	//15 minutosRefeições (Café / Almoço / Janta)xxxxxxxxxxxx
	//60 minutosRefeições (Café / Almoço / Janta)
	//10 minutosPartida de linha / Parada de Linha xxxxxxxxxxxxxx
			
	MinDispL6_1T := (((INT_TO_REAL (HoraFim1Turno) - INT_TO_REAL(HoraInicio1Turno) )*60)-
		INT_TO_REAL(MinInicio1Turno)+INT_TO_REAL(MinFim1Turno)-60-10);
		
		IF TempoProduzindoL6 < 1 THEN
			TempoProduzindoL6 :=0;
		END_IF
	
			//LÓGICA PARA VERIFICAR SE EXISTE ATRASO DE PRODUÇÃO NO INSTANTE ATUAL
		
	IF  CXS_ATRASOL6 >= 0 AND HabContL6_1T = TRUE THEN 
	CXS_ATRASOL6:= REAL_TO_INT(ProdL6_1T_realtime)-CNT_PRD_L6_1T;
	END_IF
	IF  CXS_ATRASOL6 >= 0 AND HabContL6_2T = TRUE THEN 
	CXS_ATRASOL6:= REAL_TO_INT(ProdL6_2T_realtime)-CNT_PRD_L6_1T;
	END_IF
	IF  CXS_ATRASOL6 >= 0 AND HabContL6_3T = TRUE THEN 
	CXS_ATRASOL6:=REAL_TO_INT(ProdL6_2T_realtime)-CNT_PRD_L6_1T;
	END_IF
		IF  CXS_ATRASOL6  < 0 THEN 
		CXS_ATRASOL6:= 0;
		END_IF
	
	//LÓGICA PARA VERIFICAR SE EXISTE ATRASO DE PRODUÇÃO NO INSTANTE ATUAL
		
		//LÓGICA PARA CONTAR TEMPO DE PARADA
		TempParadaL6(IN:=HabTemParadaL6 ,PT:= T#30S);
		IF TempParadaL6.Q   THEN
		TotalMinParado(IN:=HabTotalMinParado ,PT:= T#1M);
		IF TotalMinParado.Q = TRUE THEN
			TempoParadaL6 := TempoParadaL6+1;
			HabTotalMinParado := FALSE;
			ELSE
				HabTotalMinParado := TRUE;
			END_IF
		END_IF
		
		IF PULSO_CNT_L6_1T.Q = FALSE AND PULSO_CNT_L6_2T.Q = FALSE AND PULSO_CNT_L6_3T.Q = FALSE  THEN
		HabTemParadaL6 := TRUE;
		
		ELSE 	
		HabTemParadaL6 := FALSE;
		END_IF
		//LÓGICA PARA CONTAR TEMPO DE PARADA
//==============Habilita contadores 1º turno ================
IF (hora = HoraInicio1Turno AND minuto = MinInicio1Turno)  THEN
HabContL6_1T := TRUE;
HabContL6_3T := FALSE;
HabContL6_2T := FALSE;
CNT_PRD_L6_3T := 0;
CNT_PRD_L6_2T := 0;
CNT_PRD_L6_1T := 0;
TempoProduzindoL6 :=0;
EficL6_1T_projetada:=0;
EficL6_1T_realtime :=0;
ProdL6_1T_realtime :=0;
TempoParadaL6 :=0;
CXS_ATRASOL6:=0;
END_IF 


//==============Contador e Eficiencia L6 1 TURNO de cartuchos==========
IF HabContL6_1T = TRUE THEN 
PULSO_CNT_L6_1T(CLK:=CNT_L6);
//TMR_SIMUL_CNT1(IN:=LIBERA_TMR_SIMUL ,PT:=T#9S);	
		IF PULSO_CNT_L6_1T.Q = TRUE THEN
		CNT_PRD_L6_1T := CNT_PRD_L6_1T+1;
		//LIBERA_TMR_SIMUL := FALSE;
		RegistraHora := FALSE;
		MinDispTurnoAtual := MinDispL6_1T;
//ELSE 	
	//LIBERA_TMR_SIMUL:= TRUE;
		END_IF
		
			IF hora > 5 AND hora < 11 THEN

		ProdL6_1T_realtime := (INT_TO_REAL(ProducaoProgramada_L6_1T) / (MinDispL6_1T)) * ((
		(INT_TO_REAL(hora)-INT_TO_REAL(HoraInicio1Turno))*60)-INT_TO_REAL(MinInicio1Turno) + INT_TO_REAL(minuto));
		
		TempoProduzindoL6 :=  ((hora-HoraInicio1Turno)*60)-MinInicio1Turno+ minuto-TempoParadaL6;
		
		EficL6_1T_realtime := ( INT_TO_REAL(CNT_PRD_L6_1T) / ProdL6_1T_realtime ) * 100 * (EficL6_1T_projetada/100);
		EficL6_1T_projetada := (ProdL6_1T_realtime / ProducaoProgramada_L6_1T) * 100;
		END_IF
		
			IF hora > 11 AND hora < 15 THEN

		ProdL6_1T_realtime := (INT_TO_REAL(ProducaoProgramada_L6_1T) / (MinDispL6_1T)) * ((
		(INT_TO_REAL(hora)-INT_TO_REAL(HoraInicio1Turno))*60)-INT_TO_REAL(MinInicio1Turno) + INT_TO_REAL(minuto)-10-60);
		
		TempoProduzindoL6 :=  ((hora-HoraInicio1Turno)*60)-MinInicio1Turno+ minuto-TempoParadaL6;
		
		EficL6_1T_realtime := ( INT_TO_REAL(CNT_PRD_L6_1T) / ProdL6_1T_realtime ) * 100 * (EficL6_1T_projetada/100);
		EficL6_1T_projetada := (ProdL6_1T_realtime / ProducaoProgramada_L6_1T) * 100;
		END_IF
	
END_IF
EficienciaL6_1T := (INT_TO_REAL(CNT_PRD_L6_1T) / INT_TO_REAL(ProducaoProgramada_L6_1T) ) * 100;


//=====================1º TURNO ========================

//=====================2º TURNO ========================

	//10 minutos - Reunião / DSS / Treinamento
	//20 minutosPartida de linha / Parada de Linha
	//15 minutosRefeições (Café / Almoço / Janta)
	//60 minutosRefeições (Café / Almoço / Janta)
	//10 minutosPartida de linha / Parada de Linha
	IF hora = 0 THEN 
		hora := 24;
	END_IF
	
		MinDispL6_2T := (((INT_TO_REAL (HoraFim2Turno) - INT_TO_REAL(HoraInicio2Turno) )*60)-
		INT_TO_REAL(MinInicio2Turno)+INT_TO_REAL(MinFim2Turno)-60-10);
	
//==============Contador e Eficiencia L6 2 TURNO de cartuchos==========
//==============Habilita contadores 2º turno ================
IF (hora = HoraInicio2Turno AND minuto = MinInicio2Turno)  THEN
HabContL6_2T := TRUE;
HabContL6_1T := FALSE;
CNT_PRD_L6_3T := 0;
CNT_PRD_L6_2T := 0;
CNT_PRD_L6_1T := 0;
TempoParadaL6 :=0;
TempoProduzindoL6 :=0;
EficL6_1T_projetada:=0;
EficL6_1T_realtime :=0;
ProdL6_1T_realtime :=0;
TempoParadaL6 :=0;
CXS_ATRASOL6:=0;
END_IF 
IF HabContL6_2T = TRUE THEN 
PULSO_CNT_L6_2T(CLK:=CNT_L6);
//TMR_SIMUL_CNT2(IN:=LIBERA_TMR_SIMUL6T ,PT:=T#7S);
		IF PULSO_CNT_L6_2T.Q = TRUE  THEN
		CNT_PRD_L6_2T := CNT_PRD_L6_2T+1;
		//LIBERA_TMR_SIMUL6T := FALSE;
		MinDispTurnoAtual := MinDispL6_2T;
//ELSE 	
	//LIBERA_TMR_SIMUL6T:= TRUE;	
		END_IF
		CNT_PRD_L6_1T := CNT_PRD_L6_2T ;
		EficL6_1T_projetada:=EficL6_2T_projetada;
		EficL6_1T_realtime :=EficL6_2T_realtime;
		ProdL6_1T_realtime :=ProdL6_1T_realtime;
		
			IF hora > 13 AND hora < 19 THEN

		ProdL6_2T_realtime := (INT_TO_REAL(ProducaoProgramada_L6_T2) / (MinDispL6_2T)) * ((
		(INT_TO_REAL(hora)-INT_TO_REAL(HoraInicio2Turno))*60)-INT_TO_REAL(MinInicio2Turno) + INT_TO_REAL(minuto));
		
		TempoProduzindoL6 :=  ((hora-HoraInicio2Turno)*60)-MinInicio2Turno+ minuto-TempoParadaL6;
		
		EficL6_2T_realtime := ( INT_TO_REAL(CNT_PRD_L6_2T) / ProdL6_2T_realtime ) * 100 * (EficL6_2T_projetada/100);
		EficL6_2T_projetada := (ProdL6_2T_realtime / ProducaoProgramada_L6_T2) * 100;
		END_IF
		IF hora > 19 AND hora < 23 THEN

		ProdL6_2T_realtime := (INT_TO_REAL(ProducaoProgramada_L6_T2) / (MinDispL6_2T)) * ((
		(INT_TO_REAL(hora)-INT_TO_REAL(HoraInicio2Turno))*60)-INT_TO_REAL(MinInicio2Turno) + INT_TO_REAL(minuto)-10-60);
		
		TempoProduzindoL6 :=  ((hora-HoraInicio2Turno)*60)-MinInicio2Turno+ minuto-TempoParadaL6;
		
		EficL6_2T_realtime := ( INT_TO_REAL(CNT_PRD_L6_2T) / ProdL6_2T_realtime ) * 100 * (EficL6_2T_projetada/100);
		EficL6_2T_projetada := (ProdL6_2T_realtime / ProducaoProgramada_L6_T2) * 100;
		END_IF
END_IF
EficienciaL6_2T := (INT_TO_REAL (CNT_PRD_L6_2T) / INT_TO_REAL (ProducaoProgramada_L6_T2)  ) * 100;

//=====================2º TURNO ========================

//=====================3º TURNO ========================
//==============Contador e Eficiencia L6 3 TURNO de cartuchos==========

//==============Habilita contadores 3º turno ================
//10 minutos - Reunião / DSS / Treinamento
	//20 minutosPartida de linha / Parada de Linha
	//15 minutosRefeições (Café / Almoço / Janta)
	//60 minutosRefeições (Café / Almoço / Janta)
	//10 minutosPartida de linha / Parada de Linha
	IF hora = 0 THEN 
		hora := 24;
	END_IF
	
		MinDispL6_3T := (((INT_TO_REAL (HoraFim3Turno) - INT_TO_REAL(HoraInicio3Turno) )*60)-
		INT_TO_REAL(MinInicio3Turno)+INT_TO_REAL(MinFim3Turno)-60-10);
		
	
//==============Contador e Eficiencia L6 3 TURNO de cartuchos==========
//==============Habilita contadores 3º turno ================
IF (hora = HoraInicio3Turno AND minuto = MinInicio3Turno)  THEN
HabContL6_3T := TRUE;
HabContL6_2T := FALSE;
HabContL6_1T := FALSE;
CNT_PRD_L6_3T := 0;
CNT_PRD_L6_2T := 0;
CNT_PRD_L6_1T := 0;
TempoParadaL6 :=0;
TempoProduzindoL6 :=0;
EficL6_1T_projetada:=0;
EficL6_1T_realtime :=0;
ProdL6_1T_realtime :=0;
TempoParadaL6 :=0;
CXS_ATRASOL6:=0;
END_IF 

IF HabContL6_3T = TRUE THEN 
PULSO_CNT_L6_3T(CLK:=CNT_L6);	
		IF PULSO_CNT_L6_3T.Q = TRUE THEN
		CNT_PRD_L6_3T := CNT_PRD_L6_3T+1;	
			CNT_PRD_L6_1T := CNT_PRD_L6_3T ;
		EficL6_1T_projetada:=EficL6_3T_projetada;
		EficL6_1T_realtime :=EficL6_3T_realtime;
		ProdL6_1T_realtime :=ProdL6_3T_realtime;
		END_IF
		IF hora > 21 AND hora <= 24 THEN

		ProdL6_3T_realtime := (INT_TO_REAL(ProducaoProgramada_L6_T3) / (MinDispL6_3T)) * ((
		(INT_TO_REAL(hora)-INT_TO_REAL(HoraInicio3Turno))*60)-INT_TO_REAL(MinInicio3Turno) + INT_TO_REAL(minuto));
		
		TempoProduzindoL6 :=  ((hora-HoraInicio3Turno)*60)-MinInicio3Turno+ minuto-TempoParadaL6;
	
		EficL6_3T_realtime := ( INT_TO_REAL(CNT_PRD_L6_3T) / ProdL6_3T_realtime ) * 100 *(EficL6_3T_projetada/100) ;
		EficL6_3T_projetada := (ProdL6_3T_realtime / ProducaoProgramada_L6_T3) * 100;
		END_IF
		IF ((hora > 0 ) AND minuto > 30) AND hora < 2 THEN

		ProdL6_3T_realtime := (INT_TO_REAL(ProducaoProgramada_L6_T3) / (MinDispL6_3T)) * ((
		(INT_TO_REAL(hora)-INT_TO_REAL(HoraInicio3Turno))*60)-INT_TO_REAL(MinInicio3Turno) + INT_TO_REAL(minuto)-10-60);
		
		TempoProduzindoL6 :=  ((hora-HoraInicio3Turno)*60)-MinInicio3Turno+ minuto-TempoParadaL6;
	
		EficL6_3T_realtime := ( INT_TO_REAL(CNT_PRD_L6_3T) / ProdL6_3T_realtime ) * 100 *(EficL6_3T_projetada/100) ;
		EficL6_3T_projetada := (ProdL6_3T_realtime / ProducaoProgramada_L6_T3) * 100;
		END_IF
END_IF


EficienciaL6_3T := (INT_TO_REAL (CNT_PRD_L6_3T) / INT_TO_REAL (ProducaoProgramada_L6_T3)  ) * 100;


IF (hora = HoraInicio3Turno AND minuto = MinInicio3Turno)  THEN
HabContL6_3T := TRUE;
HabContL6_2T := FALSE;
END_IF 

IF HabContL6_3T = TRUE THEN 
PULSO_CNT_L6_3T(CLK:=CNT_L6);
//TMR_SIMUL_CNT3(IN:=LIBERA_TMR_SIMUL3T ,PT:=T#8S);
		IF PULSO_CNT_L6_3T.Q = TRUE  THEN
		CNT_PRD_L6_3T := CNT_PRD_L6_3T+1;
		//LIBERA_TMR_SIMUL3T := FALSE;
		MinDispTurnoAtual := MinDispL6_3T;
//ELSE 	
	//LIBERA_TMR_SIMUL3T:= TRUE;	
		END_IF
		END_IF
	
	
EficienciaL6_3T := (INT_TO_REAL (CNT_PRD_L6_3T) / INT_TO_REAL(ProducaoProgramada_L6_T3)  ) * 100;
//=====================3º TURNO ========================

IF (hora = 11 AND minuto = 0) OR (hora = 19 AND minuto = 0) OR (hora = 1 AND minuto = 30)  THEN
	refeicao := TRUE;
	END_IF
	IF (hora = 11 AND minuto = 40) OR  (hora = 20 AND minuto = 0)  OR  (hora = 2 AND minuto = 30)  THEN
	refeicao := FALSE;
	END_IF 
	
	IF (hora = 6 AND minuto = 0) OR (hora = 20 AND minuto = 0) OR (hora = 2 AND minuto = 30)  THEN
	DDS := TRUE;
	END_IF
	IF (hora = 6 AND minuto = 10) OR  (hora = 20 AND minuto = 10)  OR  (hora = 2 AND minuto = 40)  THEN
	DDS := FALSE;
	END_IF 
	IF (hora = 6 AND minuto = 0) OR (hora = 14 AND minuto = 20) OR (hora = 22 AND minuto = 30)  THEN
	SETUP := TRUE;
	END_IF
	IF (hora = 6 AND minuto = 30) OR  (hora = 14 AND minuto = 50)  OR  (hora = 23 AND minuto = 0)  THEN
	SETUP := FALSE;
	END_IF 

//STATUS DA LINHA 6
//STATUS DO EQUIPAMENTO
//0- SEM PROGRAMAÇÃO
//1- PRODUZINDO
//2- PARADA
//3- REFEIÇÃO
//4- DDS
//5- SETUP

IF ProducaoProgramada_L6_1T = 0 AND HabContL6_1T = TRUE AND TempParadaL6.Q = TRUE THEN
	Status_L6 := 0;
	L6semprogramacao :=TRUE;
	END_IF
		IF ProducaoProgramada_L6_1T > 0 AND HabContL6_1T = TRUE THEN 
		L6semprogramacao :=FALSE;
		END_IF
	
IF ProducaoProgramada_L6_T2 = 0 AND HabContL6_2T = TRUE AND TempParadaL6.Q = TRUE THEN
	Status_L6 := 0;
	L6semprogramacao :=TRUE;
		END_IF
			IF ProducaoProgramada_L6_T2 > 0 AND HabContL6_2T = TRUE THEN 
				L6semprogramacao :=FALSE;
				END_IF
				
IF ProducaoProgramada_L6_T3 = 0 AND HabContL6_3T = TRUE  AND TempParadaL6.Q = TRUE THEN
	Status_L6 := 0;
	L6semprogramacao :=TRUE;
		END_IF
			IF ProducaoProgramada_L6_T3 > 0 AND HabContL6_3T = TRUE THEN 
			L6semprogramacao :=FALSE;
			END_IF
	
IF TempParadaL6.Q = FALSE  THEN
	Status_L6 := 1;
END_IF

	IF refeicao = FALSE AND SETUP = FALSE AND DDS = FALSE AND TempParadaL6.Q = TRUE AND L6semprogramacao = FALSE THEN
	Status_L6 := 2;
	END_IF

IF refeicao = TRUE AND TempParadaL6.Q = TRUE THEN
Status_L6 := 3;
END_IF

IF DDS = TRUE AND TempParadaL6.Q = TRUE THEN
Status_L6 := 4;
END_IF

//IF SETUP = TRUE THEN
//Status_L6 := 5;
//END_IF
//STATUS DA LINHA 6

END_PROGRAM

// Device/Application/ProdL7
PROGRAM ProdL7
VAR
	//PRODUÇÃO LINHAS ENVASE
	
//=========================	
PULSO_CNT_L7_1T: R_TRIG;
PULSO_CNT_L7_2T: R_TRIG;
PULSO_CNT_L7_3T: R_TRIG;
	CNT_PRD_L7: INT;
	//CNT_L7: BOOL;
//=========================	
	Result : RTC_STATUS;
	DATEANDTIME : EXTENDED_DATE_AND_TIME;
	xEnable : BOOL;
//=========================		
	dia: INT;
	mes: INT;
	ano: INT;
	hora: INT;
	minuto: INT;
	segundo: INT;
	
	
	
	//HoraInicio1Turno: INT;
	//MinInicio1Turno: INT;
	HoraFim1Turno: INT;
	MinFim1Turno: INT;
	//HoraInicio2Turno: INT;
	//MinInicio2Turno: INT;
	HoraFim2Turno: INT;
	MinFim2Turno: INT;
	//HoraInicio3Turno: INT;
	//MinInicio3Turno: INT;
	HoraFim3Turno: INT;
	MinFim3Turno: INT;
	EficienciaL7: INT;
	
	
	HabContL7_1T: BOOL;
	HabContL7_2T: BOOL;
	HabContL7_3T: BOOL;
	
	CNT_PRD_L7_2T: INT;
	CNT_PRD_L7_3T: INT;
	EficienciaL7_1T: REAL;
	EficienciaL7_2T: REAL;
	EficienciaL7_3T: REAL;
	
	MinDispL7_1T: REAL;
	
	ProdL7_1T_realtime: REAL;
	MinDispL7_2T: REAL;
	ProdL7_2T_realtime: REAL;
	EficL7_2T_realtime: REAL;
	MinDispL7_3T: REAL;
	ProdL7_3T_realtime: REAL;
	EficL7_3T_realtime: REAL;
	
	//TMR_SIMUL_CNT1: TON;
	//LIBERA_TMR_SIMUL: BOOL;
	EficL7_2T_projetada: REAL;
	//TMR_SIMUL_CNT2: TON;
	//LIBERA_TMR_SIMUL7T: BOOL;
	//TMR_SIMUL_CNT3: TON;
	//LIBERA_TMR_SIMUL3T: BOOL;
	EficL7_3T_projetada: REAL;
//	EficL7_1T_realtime: REAL;
	HabTemParadaL7: BOOL;
	TempParadaL7: Ton;
	horaParadaL7: INT;
	MinParadaL7: INT;
	RegistraHora: BOOL;
	Borda_des_RegistraHora: F_TRIG;
	HoraRetornoParadaL7: INT;
	MinRetornoParadaL7: INT;
	TempoParadaL7L7: INT;
	TotalMinParado: TON;
	HabTotalMinParado: BOOL;
	//TempoProduzindoL7: REAL;
	//MinDispTurnoAtual: REAL;

	refeicao: BOOL;
	DDS: BOOL;
	SETUP: BOOL;
	L7semprogramacao: BOOL;
END_VAR


//LÓGICA PARA ANÁLISES DE PRODUTIVADADE DA L7 DE CARTUCHOS
	dia := BYTE_TO_INT (DATEANDTIME.byDayOfMonth);
	mes := BYTE_TO_INT (DATEANDTIME.byMonth);
	ano := WORD_TO_INT (DATEANDTIME.wYear);
	hora := BYTE_TO_INT (DATEANDTIME.byHours);
	minuto := BYTE_TO_INT (DATEANDTIME.byMinutes);
	segundo := BYTE_TO_INT (DATEANDTIME.bySeconds);
	xEnable := TRUE;
	
	//HABILITA RTC==========================
	IF xEnable = TRUE THEN
	Result := GetDateAndTime(DATEANDTIME);
	END_IF
//HABILITA RTC==========================

//=====================1º TURNO ========================
	
		//HoraInicio1Turno: INT;
	
	HoraFim1Turno:= HoraInicio2Turno;
	MinFim1Turno:= MinInicio2Turno;
	HoraFim2Turno:= HoraInicio3Turno;
	MinFim2Turno:= MinInicio3Turno;
	
	//10 minutos - Reunião / DSS / Treinamento
	//20 minutosPartida de linha / Parada de Linha xxxxxxxxxx
	//15 minutosRefeições (Café / Almoço / Janta)xxxxxxxxxxxx
	//60 minutosRefeições (Café / Almoço / Janta)
	//10 minutosPartida de linha / Parada de Linha xxxxxxxxxxxxxx
			
	MinDispL7_1T := (((INT_TO_REAL (HoraFim1Turno) - INT_TO_REAL(HoraInicio1Turno) )*60)-
		INT_TO_REAL(MinInicio1Turno)+INT_TO_REAL(MinFim1Turno)-60-10);
		
			IF TempoProduzindoL7 < 1 THEN
			TempoProduzindoL7 :=0;
		END_IF
	
		//LÓGICA PARA VERIFICAR SE EXISTE ATRASO DE PRODUÇÃO NO INSTANTE ATUAL
		
	IF  CXS_ATRASOL7 >= 0 AND HabContL7_1T = TRUE THEN 
	CXS_ATRASOL7:= REAL_TO_INT(ProdL7_1T_realtime)-CNT_PRD_L7_1T;
	END_IF
	IF  CXS_ATRASOL7 >= 0 AND HabContL7_2T = TRUE THEN 
	CXS_ATRASOL7:= REAL_TO_INT(ProdL7_2T_realtime)-CNT_PRD_L7_1T;
	END_IF
	IF  CXS_ATRASOL7 >= 0 AND HabContL7_3T = TRUE THEN 
	CXS_ATRASOL7:=REAL_TO_INT(ProdL7_2T_realtime)-CNT_PRD_L7_1T;
	END_IF
		IF  CXS_ATRASOL7  < 0 THEN 
		CXS_ATRASOL7:= 0;
		END_IF
	
	//LÓGICA PARA VERIFICAR SE EXISTE ATRASO DE PRODUÇÃO NO INSTANTE ATUAL
		
		//LÓGICA PARA CONTAR TEMPO DE PARADA
		TempParadaL7(IN:=HabTemParadaL7 ,PT:= T#30S);
		IF TempParadaL7.Q   THEN
		TotalMinParado(IN:=HabTotalMinParado ,PT:= T#1M);
		IF TotalMinParado.Q = TRUE THEN
			TempoParadaL7 := TempoParadaL7+1;
			HabTotalMinParado := FALSE;
			ELSE
				HabTotalMinParado := TRUE;
			END_IF
		END_IF
		
		IF PULSO_CNT_L7_1T.Q = FALSE AND PULSO_CNT_L7_2T.Q = FALSE AND PULSO_CNT_L7_3T.Q = FALSE  THEN
		HabTemParadaL7 := TRUE;
		
		ELSE 	
		HabTemParadaL7 := FALSE;
		END_IF
		//LÓGICA PARA CONTAR TEMPO DE PARADA
//==============Habilita contadores 1º turno ================
IF (hora = HoraInicio1Turno AND minuto = MinInicio1Turno)  THEN
HabContL7_1T := TRUE;
HabContL7_3T := FALSE;
HabContL7_2T := FALSE;
CNT_PRD_L7_3T := 0;
CNT_PRD_L7_2T := 0;
CNT_PRD_L7_1T := 0;
TempoProduzindoL7 :=0;
EficL7_1T_projetada:=0;
EficL7_1T_realtime :=0;
ProdL7_1T_realtime :=0;
TempoParadaL7 :=0;
CXS_ATRASOL1:=0;
END_IF 


//==============Contador e Eficiencia L7 1 TURNO de cartuchos==========
IF HabContL7_1T = TRUE THEN 
PULSO_CNT_L7_1T(CLK:=CNT_L7);
//TMR_SIMUL_CNT1(IN:=LIBERA_TMR_SIMUL ,PT:=T#9S);	
		IF PULSO_CNT_L7_1T.Q = TRUE THEN
		CNT_PRD_L7_1T := CNT_PRD_L7_1T+1;
		//LIBERA_TMR_SIMUL := FALSE;
		RegistraHora := FALSE;
		MinDispTurnoAtual := MinDispL7_1T;
//ELSE 	
	//LIBERA_TMR_SIMUL:= TRUE;
		END_IF
		
			IF hora > 5 AND hora < 11 THEN

		ProdL7_1T_realtime := (INT_TO_REAL(ProducaoProgramada_L7_1T) / (MinDispL7_1T)) * ((
		(INT_TO_REAL(hora)-INT_TO_REAL(HoraInicio1Turno))*60)-INT_TO_REAL(MinInicio1Turno) + INT_TO_REAL(minuto));
		
		TempoProduzindoL7 :=  ((hora-HoraInicio1Turno)*60)-MinInicio1Turno+ minuto-TempoParadaL7;
		
		EficL7_1T_realtime := ( INT_TO_REAL(CNT_PRD_L7_1T) / ProdL7_1T_realtime ) * 100 * (EficL7_1T_projetada/100);
		EficL7_1T_projetada := (ProdL7_1T_realtime / ProducaoProgramada_L7_1T) * 100;
		END_IF
		
			IF hora > 11 AND hora < 15 THEN

		ProdL7_1T_realtime := (INT_TO_REAL(ProducaoProgramada_L7_1T) / (MinDispL7_1T)) * ((
		(INT_TO_REAL(hora)-INT_TO_REAL(HoraInicio1Turno))*60)-INT_TO_REAL(MinInicio1Turno) + INT_TO_REAL(minuto)-10-60);
		
		TempoProduzindoL7 :=  ((hora-HoraInicio1Turno)*60)-MinInicio1Turno+ minuto-TempoParadaL7;
		
		EficL7_1T_realtime := ( INT_TO_REAL(CNT_PRD_L7_1T) / ProdL7_1T_realtime ) * 100 * (EficL7_1T_projetada/100);
		EficL7_1T_projetada := (ProdL7_1T_realtime / ProducaoProgramada_L7_1T) * 100;
		END_IF
	
END_IF
EficienciaL7_1T := (INT_TO_REAL(CNT_PRD_L7_1T) / INT_TO_REAL(ProducaoProgramada_L7_1T) ) * 100;


//=====================1º TURNO ========================

//=====================2º TURNO ========================

	//10 minutos - Reunião / DSS / Treinamento
	//20 minutosPartida de linha / Parada de Linha
	//15 minutosRefeições (Café / Almoço / Janta)
	//60 minutosRefeições (Café / Almoço / Janta)
	//10 minutosPartida de linha / Parada de Linha
	IF hora = 0 THEN 
		hora := 24;
	END_IF
	
		MinDispL7_2T := (((INT_TO_REAL (HoraFim2Turno) - INT_TO_REAL(HoraInicio2Turno) )*60)-
		INT_TO_REAL(MinInicio2Turno)+INT_TO_REAL(MinFim2Turno)-60-10);
	
//==============Contador e Eficiencia L7 2 TURNO de cartuchos==========
//==============Habilita contadores 2º turno ================
IF (hora = HoraInicio2Turno AND minuto = MinInicio2Turno)  THEN
HabContL7_2T := TRUE;
HabContL7_1T := FALSE;
CNT_PRD_L7_3T := 0;
CNT_PRD_L7_2T := 0;
CNT_PRD_L7_1T := 0;
TempoParadaL7 :=0;
TempoProduzindoL7 :=0;
EficL7_1T_projetada:=0;
EficL7_1T_realtime :=0;
ProdL7_1T_realtime :=0;
TempoParadaL7 :=0;
CXS_ATRASOL1:=0;
END_IF 
IF HabContL7_2T = TRUE THEN 
PULSO_CNT_L7_2T(CLK:=CNT_L7);
//TMR_SIMUL_CNT2(IN:=LIBERA_TMR_SIMUL7T ,PT:=T#7S);
		IF PULSO_CNT_L7_2T.Q = TRUE  THEN
		CNT_PRD_L7_2T := CNT_PRD_L7_2T+1;
		//LIBERA_TMR_SIMUL7T := FALSE;
		MinDispTurnoAtual := MinDispL7_2T;
//ELSE 	
	//LIBERA_TMR_SIMUL7T:= TRUE;	
		END_IF
		CNT_PRD_L7_1T := CNT_PRD_L7_2T ;
		EficL7_1T_projetada:=EficL7_2T_projetada;
		EficL7_1T_realtime :=EficL7_2T_realtime;
		ProdL7_1T_realtime :=ProdL7_1T_realtime;
		
			IF hora > 13 AND hora < 19 THEN

		ProdL7_2T_realtime := (INT_TO_REAL(ProducaoProgramada_L7_T2) / (MinDispL7_2T)) * ((
		(INT_TO_REAL(hora)-INT_TO_REAL(HoraInicio2Turno))*60)-INT_TO_REAL(MinInicio2Turno) + INT_TO_REAL(minuto));
		
		TempoProduzindoL7 :=  ((hora-HoraInicio2Turno)*60)-MinInicio2Turno+ minuto-TempoParadaL7;
		
		EficL7_2T_realtime := ( INT_TO_REAL(CNT_PRD_L7_2T) / ProdL7_2T_realtime ) * 100 * (EficL7_2T_projetada/100);
		EficL7_2T_projetada := (ProdL7_2T_realtime / ProducaoProgramada_L7_T2) * 100;
		END_IF
		IF hora > 19 AND hora < 23 THEN

		ProdL7_2T_realtime := (INT_TO_REAL(ProducaoProgramada_L7_T2) / (MinDispL7_2T)) * ((
		(INT_TO_REAL(hora)-INT_TO_REAL(HoraInicio2Turno))*60)-INT_TO_REAL(MinInicio2Turno) + INT_TO_REAL(minuto)-10-60);
		
		TempoProduzindoL7 :=  ((hora-HoraInicio2Turno)*60)-MinInicio2Turno+ minuto-TempoParadaL7;
		
		EficL7_2T_realtime := ( INT_TO_REAL(CNT_PRD_L7_2T) / ProdL7_2T_realtime ) * 100 * (EficL7_2T_projetada/100);
		EficL7_2T_projetada := (ProdL7_2T_realtime / ProducaoProgramada_L7_T2) * 100;
		END_IF
END_IF
EficienciaL7_2T := (INT_TO_REAL (CNT_PRD_L7_2T) / INT_TO_REAL (ProducaoProgramada_L7_T2)  ) * 100;

//=====================2º TURNO ========================

//=====================3º TURNO ========================
//==============Contador e Eficiencia L7 3 TURNO de cartuchos==========

//==============Habilita contadores 3º turno ================
//10 minutos - Reunião / DSS / Treinamento
	//20 minutosPartida de linha / Parada de Linha
	//15 minutosRefeições (Café / Almoço / Janta)
	//60 minutosRefeições (Café / Almoço / Janta)
	//10 minutosPartida de linha / Parada de Linha
	IF hora = 0 THEN 
		hora := 24;
	END_IF
	
		MinDispL7_3T := (((INT_TO_REAL (HoraFim3Turno) - INT_TO_REAL(HoraInicio3Turno) )*60)-
		INT_TO_REAL(MinInicio3Turno)+INT_TO_REAL(MinFim3Turno)-60-10);
		
	
//==============Contador e Eficiencia L7 3 TURNO de cartuchos==========
//==============Habilita contadores 3º turno ================
IF (hora = HoraInicio3Turno AND minuto = MinInicio3Turno)  THEN
HabContL7_3T := TRUE;
HabContL7_2T := FALSE;
HabContL7_1T := FALSE;
CNT_PRD_L7_3T := 0;
CNT_PRD_L7_2T := 0;
CNT_PRD_L7_1T := 0;
TempoParadaL7 :=0;
TempoProduzindoL7 :=0;
EficL7_1T_projetada:=0;
EficL7_1T_realtime :=0;
ProdL7_1T_realtime :=0;
TempoParadaL7 :=0;
END_IF 

IF HabContL7_3T = TRUE THEN 
PULSO_CNT_L7_3T(CLK:=CNT_L7);	
		IF PULSO_CNT_L7_3T.Q = TRUE THEN
		CNT_PRD_L7_3T := CNT_PRD_L7_3T+1;	
			CNT_PRD_L7_1T := CNT_PRD_L7_3T ;
		EficL7_1T_projetada:=EficL7_3T_projetada;
		EficL7_1T_realtime :=EficL7_3T_realtime;
		ProdL7_1T_realtime :=ProdL7_3T_realtime;
		END_IF
		IF hora > 21 AND hora <= 24 THEN

		ProdL7_3T_realtime := (INT_TO_REAL(ProducaoProgramada_L7_T3) / (MinDispL7_3T)) * ((
		(INT_TO_REAL(hora)-INT_TO_REAL(HoraInicio3Turno))*60)-INT_TO_REAL(MinInicio3Turno) + INT_TO_REAL(minuto));
		
		TempoProduzindoL7 :=  ((hora-HoraInicio3Turno)*60)-MinInicio3Turno+ minuto-TempoParadaL7;
	
		EficL7_3T_realtime := ( INT_TO_REAL(CNT_PRD_L7_3T) / ProdL7_3T_realtime ) * 100 *(EficL7_3T_projetada/100) ;
		EficL7_3T_projetada := (ProdL7_3T_realtime / ProducaoProgramada_L7_T3) * 100;
		END_IF
		IF ((hora > 0 ) AND minuto > 30) AND hora < 2 THEN

		ProdL7_3T_realtime := (INT_TO_REAL(ProducaoProgramada_L7_T3) / (MinDispL7_3T)) * ((
		(INT_TO_REAL(hora)-INT_TO_REAL(HoraInicio3Turno))*60)-INT_TO_REAL(MinInicio3Turno) + INT_TO_REAL(minuto)-10-60);
		
		TempoProduzindoL7 :=  ((hora-HoraInicio3Turno)*60)-MinInicio3Turno+ minuto-TempoParadaL7;
	
		EficL7_3T_realtime := ( INT_TO_REAL(CNT_PRD_L7_3T) / ProdL7_3T_realtime ) * 100 *(EficL7_3T_projetada/100) ;
		EficL7_3T_projetada := (ProdL7_3T_realtime / ProducaoProgramada_L7_T3) * 100;
		END_IF
END_IF


EficienciaL7_3T := (INT_TO_REAL (CNT_PRD_L7_3T) / INT_TO_REAL (ProducaoProgramada_L7_T3)  ) * 100;


IF (hora = HoraInicio3Turno AND minuto = MinInicio3Turno)  THEN
HabContL7_3T := TRUE;
HabContL7_2T := FALSE;
END_IF 

IF HabContL7_3T = TRUE THEN 
PULSO_CNT_L7_3T(CLK:=CNT_L7);
//TMR_SIMUL_CNT3(IN:=LIBERA_TMR_SIMUL3T ,PT:=T#8S);
		IF PULSO_CNT_L7_3T.Q = TRUE  THEN
		CNT_PRD_L7_3T := CNT_PRD_L7_3T+1;
		//LIBERA_TMR_SIMUL3T := FALSE;
		MinDispTurnoAtual := MinDispL7_3T;
//ELSE 	
	//LIBERA_TMR_SIMUL3T:= TRUE;	
		END_IF
		END_IF
	
	
EficienciaL7_3T := (INT_TO_REAL (CNT_PRD_L7_3T) / INT_TO_REAL(ProducaoProgramada_L7_T3)  ) * 100;
//=====================3º TURNO ========================

IF (hora = 11 AND minuto = 0) OR (hora = 19 AND minuto = 0) OR (hora = 1 AND minuto = 30)  THEN
	refeicao := TRUE;
	END_IF
	IF (hora = 11 AND minuto = 40) OR  (hora = 20 AND minuto = 0)  OR  (hora = 2 AND minuto = 30)  THEN
	refeicao := FALSE;
	END_IF 
	
	IF (hora = 6 AND minuto = 0) OR (hora = 20 AND minuto = 0) OR (hora = 2 AND minuto = 30)  THEN
	DDS := TRUE;
	END_IF
	IF (hora = 6 AND minuto = 10) OR  (hora = 20 AND minuto = 10)  OR  (hora = 2 AND minuto = 40)  THEN
	DDS := FALSE;
	END_IF 
	IF (hora = 6 AND minuto = 0) OR (hora = 14 AND minuto = 20) OR (hora = 22 AND minuto = 30)  THEN
	SETUP := TRUE;
	END_IF
	IF (hora = 6 AND minuto = 30) OR  (hora = 14 AND minuto = 50)  OR  (hora = 23 AND minuto = 0)  THEN
	SETUP := FALSE;
	END_IF 

//STATUS DA LINHA 7
//STATUS DO EQUIPAMENTO
//0- SEM PROGRAMAÇÃO
//1- PRODUZINDO
//2- PARADA
//3- REFEIÇÃO
//4- DDS
//5- SETUP

IF ProducaoProgramada_L7_1T = 0 AND HabContL7_1T = TRUE AND TempParadaL7.Q = TRUE THEN
	Status_L7 := 0;
	L7semprogramacao :=TRUE;
	END_IF
		IF ProducaoProgramada_L7_1T > 0 AND HabContL7_1T = TRUE THEN 
		L7semprogramacao :=FALSE;
		END_IF
	
IF ProducaoProgramada_L7_T2 = 0 AND HabContL7_2T = TRUE AND TempParadaL7.Q = TRUE THEN
	Status_L7 := 0;
	L7semprogramacao :=TRUE;
		END_IF
			IF ProducaoProgramada_L7_T2 > 0 AND HabContL7_2T = TRUE THEN 
				L7semprogramacao :=FALSE;
				END_IF
				
IF ProducaoProgramada_L7_T3 = 0 AND HabContL7_3T = TRUE AND TempParadaL7.Q = TRUE THEN
	Status_L7 := 0;
	L7semprogramacao :=TRUE;
		END_IF
			IF ProducaoProgramada_L7_T3 > 0 AND HabContL7_3T = TRUE THEN 
			L7semprogramacao :=FALSE;
			END_IF
	
IF TempParadaL7.Q = FALSE THEN
	Status_L7 := 1;
END_IF

	IF refeicao = FALSE AND SETUP = FALSE AND DDS = FALSE AND TempParadaL7.Q = TRUE AND L7semprogramacao = FALSE THEN
	Status_L7 := 2;
	END_IF

IF refeicao = TRUE AND TempParadaL7.Q = TRUE THEN
Status_L7 := 3;
END_IF

IF DDS = TRUE AND TempParadaL7.Q = TRUE THEN
Status_L7 := 4;
END_IF

//IF SETUP = TRUE THEN
//Status_L7 := 5;
//END_IF
//STATUS DA LINHA 7

END_PROGRAM

// Device/Application/ProdL8
PROGRAM ProdL8
VAR
	//PRODUÇÃO LINHAS ENVASE
	
//=========================	
PULSO_CNT_L8_1T: R_TRIG;
PULSO_CNT_L8_2T: R_TRIG;
PULSO_CNT_L8_3T: R_TRIG;
	CNT_PRD_L8: INT;
	//CNT_L8: BOOL;
//=========================	
	Result : RTC_STATUS;
	DATEANDTIME : EXTENDED_DATE_AND_TIME;
	xEnable : BOOL;
//=========================		
	dia: INT;
	mes: INT;
	ano: INT;
	hora: INT;
	minuto: INT;
	segundo: INT;
	
	
	
	//HoraInicio1Turno: INT;
	//MinInicio1Turno: INT;
	HoraFim1Turno: INT;
	MinFim1Turno: INT;
	//HoraInicio2Turno: INT;
	//MinInicio2Turno: INT;
	HoraFim2Turno: INT;
	MinFim2Turno: INT;
	//HoraInicio3Turno: INT;
	//MinInicio3Turno: INT;
	HoraFim3Turno: INT;
	MinFim3Turno: INT;
	EficienciaL8: INT;
	
	
	HabContL8_1T: BOOL;
	HabContL8_2T: BOOL;
	HabContL8_3T: BOOL;
	
	CNT_PRD_L8_2T: INT;
	CNT_PRD_L8_3T: INT;
	EficienciaL8_1T: REAL;
	EficienciaL8_2T: REAL;
	EficienciaL8_3T: REAL;
	
	MinDispL8_1T: REAL;
	
	ProdL8_1T_realtime: REAL;
	MinDispL8_2T: REAL;
	ProdL8_2T_realtime: REAL;
	EficL8_2T_realtime: REAL;
	MinDispL8_3T: REAL;
	ProdL8_3T_realtime: REAL;
	EficL8_3T_realtime: REAL;
	
	//TMR_SIMUL_CNT1: TON;
	//LIBERA_TMR_SIMUL: BOOL;
	EficL8_2T_projetada: REAL;
	//TMR_SIMUL_CNT2: TON;
	//LIBERA_TMR_SIMUL8T: BOOL;
	//TMR_SIMUL_CNT3: TON;
	//LIBERA_TMR_SIMUL3T: BOOL;
	EficL8_3T_projetada: REAL;
//	EficL8_1T_realtime: REAL;
	HabTemParadaL8: BOOL;
	TempParadaL8: Ton;
	horaParadaL8: INT;
	MinParadaL8: INT;
	RegistraHora: BOOL;
	Borda_des_RegistraHora: F_TRIG;
	HoraRetornoParadaL8: INT;
	MinRetornoParadaL8: INT;
	TempoParadaL8L8: INT;
	TotalMinParado: TON;
	HabTotalMinParado: BOOL;
	//TempoProduzindoL8: REAL;
	//MinDispTurnoAtual: REAL;

	refeicao: BOOL;
	DDS: BOOL;
	SETUP: BOOL;
	L8semprogramacao: BOOL;
END_VAR


//LÓGICA PARA ANÁLISES DE PRODUTIVADADE DA L8 DE CARTUCHOS
	dia := BYTE_TO_INT (DATEANDTIME.byDayOfMonth);
	mes := BYTE_TO_INT (DATEANDTIME.byMonth);
	ano := WORD_TO_INT (DATEANDTIME.wYear);
	hora := BYTE_TO_INT (DATEANDTIME.byHours);
	minuto := BYTE_TO_INT (DATEANDTIME.byMinutes);
	segundo := BYTE_TO_INT (DATEANDTIME.bySeconds);
	xEnable := TRUE;
	
	//HABILITA RTC==========================
	IF xEnable = TRUE THEN
	Result := GetDateAndTime(DATEANDTIME);
	END_IF
//HABILITA RTC==========================

//=====================1º TURNO ========================
	
		//HoraInicio1Turno: INT;
	
	HoraFim1Turno:= HoraInicio2Turno;
	MinFim1Turno:= MinInicio2Turno;
	HoraFim2Turno:= HoraInicio3Turno;
	MinFim2Turno:= MinInicio3Turno;
	
	//10 minutos - Reunião / DSS / Treinamento
	//20 minutosPartida de linha / Parada de Linha xxxxxxxxxx
	//15 minutosRefeições (Café / Almoço / Janta)xxxxxxxxxxxx
	//60 minutosRefeições (Café / Almoço / Janta)
	//10 minutosPartida de linha / Parada de Linha xxxxxxxxxxxxxx
			
	MinDispL8_1T := (((INT_TO_REAL (HoraFim1Turno) - INT_TO_REAL(HoraInicio1Turno) )*60)-
		INT_TO_REAL(MinInicio1Turno)+INT_TO_REAL(MinFim1Turno)-60-10);
		
			IF TempoProduzindoL8 < 1 THEN
			TempoProduzindoL8 :=0;
		END_IF
	
		//LÓGICA PARA VERIFICAR SE EXISTE ATRASO DE PRODUÇÃO NO INSTANTE ATUAL
		
	IF  CXS_ATRASOL8 >= 0 AND HabContL8_1T = TRUE THEN 
	CXS_ATRASOL8:= REAL_TO_INT(ProdL8_1T_realtime)-CNT_PRD_L8_1T;
	END_IF
	IF  CXS_ATRASOL8 >= 0 AND HabContL8_2T = TRUE THEN 
	CXS_ATRASOL8:= REAL_TO_INT(ProdL8_2T_realtime)-CNT_PRD_L8_1T;
	END_IF
	IF  CXS_ATRASOL8 >= 0 AND HabContL8_3T = TRUE THEN 
	CXS_ATRASOL8:=REAL_TO_INT(ProdL8_2T_realtime)-CNT_PRD_L8_1T;
	END_IF
		IF  CXS_ATRASOL8  < 0 THEN 
		CXS_ATRASOL8:= 0;
		END_IF
	
	//LÓGICA PARA VERIFICAR SE EXISTE ATRASO DE PRODUÇÃO NO INSTANTE ATUAL
		
		//LÓGICA PARA CONTAR TEMPO DE PARADA
		TempParadaL8(IN:=HabTemParadaL8 ,PT:= T#30S);
		IF TempParadaL8.Q   THEN
		TotalMinParado(IN:=HabTotalMinParado ,PT:= T#1M);
		IF TotalMinParado.Q = TRUE THEN
			TempoParadaL8 := TempoParadaL8+1;
			HabTotalMinParado := FALSE;
			ELSE
				HabTotalMinParado := TRUE;
			END_IF
		END_IF
		
		IF PULSO_CNT_L8_1T.Q = FALSE AND PULSO_CNT_L8_2T.Q = FALSE AND PULSO_CNT_L8_3T.Q = FALSE  THEN
		HabTemParadaL8 := TRUE;
		
		ELSE 	
		HabTemParadaL8 := FALSE;
		END_IF
		//LÓGICA PARA CONTAR TEMPO DE PARADA
//==============Habilita contadores 1º turno ================
IF (hora = HoraInicio1Turno AND minuto = MinInicio1Turno)  THEN
HabContL8_1T := TRUE;
HabContL8_3T := FALSE;
HabContL8_2T := FALSE;
CNT_PRD_L8_3T := 0;
CNT_PRD_L8_2T := 0;
CNT_PRD_L8_1T := 0;
TempoProduzindoL8 :=0;
EficL8_1T_projetada:=0;
EficL8_1T_realtime :=0;
ProdL8_1T_realtime :=0;
TempoParadaL8 :=0;
CXS_ATRASOL8:=0;
END_IF 


//==============Contador e Eficiencia L8 1 TURNO de cartuchos==========
IF HabContL8_1T = TRUE THEN 
PULSO_CNT_L8_1T(CLK:=CNT_L8);
//TMR_SIMUL_CNT1(IN:=LIBERA_TMR_SIMUL ,PT:=T#9S);	
		IF PULSO_CNT_L8_1T.Q = TRUE THEN
		CNT_PRD_L8_1T := CNT_PRD_L8_1T+1;
		//LIBERA_TMR_SIMUL := FALSE;
		RegistraHora := FALSE;
		MinDispTurnoAtual := MinDispL8_1T;
//ELSE 	
	//LIBERA_TMR_SIMUL:= TRUE;
		END_IF
		
			IF hora > 5 AND hora < 11 THEN

		ProdL8_1T_realtime := (INT_TO_REAL(ProducaoProgramada_L8_1T) / (MinDispL8_1T)) * ((
		(INT_TO_REAL(hora)-INT_TO_REAL(HoraInicio1Turno))*60)-INT_TO_REAL(MinInicio1Turno) + INT_TO_REAL(minuto));
		
		TempoProduzindoL8 :=  ((hora-HoraInicio1Turno)*60)-MinInicio1Turno+ minuto-TempoParadaL8;
		
		EficL8_1T_realtime := ( INT_TO_REAL(CNT_PRD_L8_1T) / ProdL8_1T_realtime ) * 100 * (EficL8_1T_projetada/100);
		EficL8_1T_projetada := (ProdL8_1T_realtime / ProducaoProgramada_L8_1T) * 100;
		END_IF
		
			IF hora > 11 AND hora < 15 THEN

		ProdL8_1T_realtime := (INT_TO_REAL(ProducaoProgramada_L8_1T) / (MinDispL8_1T)) * ((
		(INT_TO_REAL(hora)-INT_TO_REAL(HoraInicio1Turno))*60)-INT_TO_REAL(MinInicio1Turno) + INT_TO_REAL(minuto)-10-60);
		
		TempoProduzindoL8 :=  ((hora-HoraInicio1Turno)*60)-MinInicio1Turno+ minuto-TempoParadaL8;
		
		EficL8_1T_realtime := ( INT_TO_REAL(CNT_PRD_L8_1T) / ProdL8_1T_realtime ) * 100 * (EficL8_1T_projetada/100);
		EficL8_1T_projetada := (ProdL8_1T_realtime / ProducaoProgramada_L8_1T) * 100;
		END_IF
	
END_IF
EficienciaL8_1T := (INT_TO_REAL(CNT_PRD_L8_1T) / INT_TO_REAL(ProducaoProgramada_L8_1T) ) * 100;


//=====================1º TURNO ========================

//=====================2º TURNO ========================

	//10 minutos - Reunião / DSS / Treinamento
	//20 minutosPartida de linha / Parada de Linha
	//15 minutosRefeições (Café / Almoço / Janta)
	//60 minutosRefeições (Café / Almoço / Janta)
	//10 minutosPartida de linha / Parada de Linha
	IF hora = 0 THEN 
		hora := 24;
	END_IF
	
		MinDispL8_2T := (((INT_TO_REAL (HoraFim2Turno) - INT_TO_REAL(HoraInicio2Turno) )*60)-
		INT_TO_REAL(MinInicio2Turno)+INT_TO_REAL(MinFim2Turno)-60-10);
	
//==============Contador e Eficiencia L8 2 TURNO de cartuchos==========
//==============Habilita contadores 2º turno ================
IF (hora = HoraInicio2Turno AND minuto = MinInicio2Turno)  THEN
HabContL8_2T := TRUE;
HabContL8_1T := FALSE;
CNT_PRD_L8_3T := 0;
CNT_PRD_L8_2T := 0;
CNT_PRD_L8_1T := 0;
TempoParadaL8 :=0;
TempoProduzindoL8 :=0;
EficL8_1T_projetada:=0;
EficL8_1T_realtime :=0;
ProdL8_1T_realtime :=0;
TempoParadaL8 :=0;
CXS_ATRASOL8:=0;
END_IF 
IF HabContL8_2T = TRUE THEN 
PULSO_CNT_L8_2T(CLK:=CNT_L8);
//TMR_SIMUL_CNT2(IN:=LIBERA_TMR_SIMUL8T ,PT:=T#7S);
		IF PULSO_CNT_L8_2T.Q = TRUE  THEN
		CNT_PRD_L8_2T := CNT_PRD_L8_2T+1;
		//LIBERA_TMR_SIMUL8T := FALSE;
		MinDispTurnoAtual := MinDispL8_2T;
//ELSE 	
	//LIBERA_TMR_SIMUL8T:= TRUE;	
		END_IF
		CNT_PRD_L8_1T := CNT_PRD_L8_2T ;
		EficL8_1T_projetada:=EficL8_2T_projetada;
		EficL8_1T_realtime :=EficL8_2T_realtime;
		ProdL8_1T_realtime :=ProdL8_1T_realtime;
		
			IF hora > 13 AND hora < 19 THEN

		ProdL8_2T_realtime := (INT_TO_REAL(ProducaoProgramada_L8_T2) / (MinDispL8_2T)) * ((
		(INT_TO_REAL(hora)-INT_TO_REAL(HoraInicio2Turno))*60)-INT_TO_REAL(MinInicio2Turno) + INT_TO_REAL(minuto));
		
		TempoProduzindoL8 :=  ((hora-HoraInicio2Turno)*60)-MinInicio2Turno+ minuto-TempoParadaL8;
		
		EficL8_2T_realtime := ( INT_TO_REAL(CNT_PRD_L8_2T) / ProdL8_2T_realtime ) * 100 * (EficL8_2T_projetada/100);
		EficL8_2T_projetada := (ProdL8_2T_realtime / ProducaoProgramada_L8_T2) * 100;
		END_IF
		IF hora > 19 AND hora < 23 THEN

		ProdL8_2T_realtime := (INT_TO_REAL(ProducaoProgramada_L8_T2) / (MinDispL8_2T)) * ((
		(INT_TO_REAL(hora)-INT_TO_REAL(HoraInicio2Turno))*60)-INT_TO_REAL(MinInicio2Turno) + INT_TO_REAL(minuto)-10-60);
		
		TempoProduzindoL8 :=  ((hora-HoraInicio2Turno)*60)-MinInicio2Turno+ minuto-TempoParadaL8;
		
		EficL8_2T_realtime := ( INT_TO_REAL(CNT_PRD_L8_2T) / ProdL8_2T_realtime ) * 100 * (EficL8_2T_projetada/100);
		EficL8_2T_projetada := (ProdL8_2T_realtime / ProducaoProgramada_L8_T2) * 100;
		END_IF
END_IF
EficienciaL8_2T := (INT_TO_REAL (CNT_PRD_L8_2T) / INT_TO_REAL (ProducaoProgramada_L8_T2)  ) * 100;

//=====================2º TURNO ========================

//=====================3º TURNO ========================
//==============Contador e Eficiencia L8 3 TURNO de cartuchos==========

//==============Habilita contadores 3º turno ================
//10 minutos - Reunião / DSS / Treinamento
	//20 minutosPartida de linha / Parada de Linha
	//15 minutosRefeições (Café / Almoço / Janta)
	//60 minutosRefeições (Café / Almoço / Janta)
	//10 minutosPartida de linha / Parada de Linha
	IF hora = 0 THEN 
		hora := 24;
	END_IF
	
		MinDispL8_3T := (((INT_TO_REAL (HoraFim3Turno) - INT_TO_REAL(HoraInicio3Turno) )*60)-
		INT_TO_REAL(MinInicio3Turno)+INT_TO_REAL(MinFim3Turno)-60-10);
		
	
//==============Contador e Eficiencia L8 3 TURNO de cartuchos==========
//==============Habilita contadores 3º turno ================
IF (hora = HoraInicio3Turno AND minuto = MinInicio3Turno)  THEN
HabContL8_3T := TRUE;
HabContL8_2T := FALSE;
HabContL8_1T := FALSE;
CNT_PRD_L8_3T := 0;
CNT_PRD_L8_2T := 0;
CNT_PRD_L8_1T := 0;
TempoParadaL8 :=0;
TempoProduzindoL8 :=0;
EficL8_1T_projetada:=0;
EficL8_1T_realtime :=0;
ProdL8_1T_realtime :=0;
TempoParadaL8 :=0;
CXS_ATRASOL8:=0;
END_IF 

IF HabContL8_3T = TRUE THEN 
PULSO_CNT_L8_3T(CLK:=CNT_L8);	
		IF PULSO_CNT_L8_3T.Q = TRUE THEN
		CNT_PRD_L8_3T := CNT_PRD_L8_3T+1;	
			CNT_PRD_L8_1T := CNT_PRD_L8_3T ;
		EficL8_1T_projetada:=EficL8_3T_projetada;
		EficL8_1T_realtime :=EficL8_3T_realtime;
		ProdL8_1T_realtime :=ProdL8_3T_realtime;
		END_IF
		IF hora > 21 AND hora <= 24 THEN

		ProdL8_3T_realtime := (INT_TO_REAL(ProducaoProgramada_L8_T3) / (MinDispL8_3T)) * ((
		(INT_TO_REAL(hora)-INT_TO_REAL(HoraInicio3Turno))*60)-INT_TO_REAL(MinInicio3Turno) + INT_TO_REAL(minuto));
		
		TempoProduzindoL8 :=  ((hora-HoraInicio3Turno)*60)-MinInicio3Turno+ minuto-TempoParadaL8;
	
		EficL8_3T_realtime := ( INT_TO_REAL(CNT_PRD_L8_3T) / ProdL8_3T_realtime ) * 100 *(EficL8_3T_projetada/100) ;
		EficL8_3T_projetada := (ProdL8_3T_realtime / ProducaoProgramada_L8_T3) * 100;
		END_IF
		IF ((hora > 0 ) AND minuto > 30) AND hora < 2 THEN

		ProdL8_3T_realtime := (INT_TO_REAL(ProducaoProgramada_L8_T3) / (MinDispL8_3T)) * ((
		(INT_TO_REAL(hora)-INT_TO_REAL(HoraInicio3Turno))*60)-INT_TO_REAL(MinInicio3Turno) + INT_TO_REAL(minuto)-10-60);
		
		TempoProduzindoL8 :=  ((hora-HoraInicio3Turno)*60)-MinInicio3Turno+ minuto-TempoParadaL8;
	
		EficL8_3T_realtime := ( INT_TO_REAL(CNT_PRD_L8_3T) / ProdL8_3T_realtime ) * 100 *(EficL8_3T_projetada/100) ;
		EficL8_3T_projetada := (ProdL8_3T_realtime / ProducaoProgramada_L8_T3) * 100;
		END_IF
END_IF


EficienciaL8_3T := (INT_TO_REAL (CNT_PRD_L8_3T) / INT_TO_REAL (ProducaoProgramada_L8_T3)  ) * 100;


IF (hora = HoraInicio3Turno AND minuto = MinInicio3Turno)  THEN
HabContL8_3T := TRUE;
HabContL8_2T := FALSE;
END_IF 

IF HabContL8_3T = TRUE THEN 
PULSO_CNT_L8_3T(CLK:=CNT_L8);
//TMR_SIMUL_CNT3(IN:=LIBERA_TMR_SIMUL3T ,PT:=T#8S);
		IF PULSO_CNT_L8_3T.Q = TRUE  THEN
		CNT_PRD_L8_3T := CNT_PRD_L8_3T+1;
		//LIBERA_TMR_SIMUL3T := FALSE;
		MinDispTurnoAtual := MinDispL8_3T;
//ELSE 	
	//LIBERA_TMR_SIMUL3T:= TRUE;	
		END_IF
		END_IF
	
	
EficienciaL8_3T := (INT_TO_REAL (CNT_PRD_L8_3T) / INT_TO_REAL(ProducaoProgramada_L8_T3)  ) * 100;
//=====================3º TURNO ========================

IF (hora = 11 AND minuto = 0) OR (hora = 19 AND minuto = 0) OR (hora = 1 AND minuto = 30)  THEN
	refeicao := TRUE;
	END_IF
	IF (hora = 11 AND minuto = 40) OR  (hora = 20 AND minuto = 0)  OR  (hora = 2 AND minuto = 30)  THEN
	refeicao := FALSE;
	END_IF 
	
	IF (hora = 6 AND minuto = 0) OR (hora = 20 AND minuto = 0) OR (hora = 2 AND minuto = 30)  THEN
	DDS := TRUE;
	END_IF
	IF (hora = 6 AND minuto = 10) OR  (hora = 20 AND minuto = 10)  OR  (hora = 2 AND minuto = 40)  THEN
	DDS := FALSE;
	END_IF 
	IF (hora = 6 AND minuto = 0) OR (hora = 14 AND minuto = 20) OR (hora = 22 AND minuto = 30)  THEN
	SETUP := TRUE;
	END_IF
	IF (hora = 6 AND minuto = 30) OR  (hora = 14 AND minuto = 50)  OR  (hora = 23 AND minuto = 0)  THEN
	SETUP := FALSE;
	END_IF 

//STATUS DA LINHA 8
//STATUS DO EQUIPAMENTO
//0- SEM PROGRAMAÇÃO
//1- PRODUZINDO
//2- PARADA
//3- REFEIÇÃO
//4- DDS
//5- SETUP

IF ProducaoProgramada_L8_1T = 0 AND HabContL8_1T = TRUE AND TempParadaL8.Q = TRUE THEN
	Status_L8 := 0;
	L8semprogramacao :=TRUE;
	END_IF
		IF ProducaoProgramada_L8_1T > 0 AND HabContL8_1T = TRUE THEN 
		L8semprogramacao :=FALSE;
		END_IF
	
IF ProducaoProgramada_L8_T2 = 0 AND HabContL8_2T = TRUE AND TempParadaL8.Q = TRUE THEN
	Status_L8 := 0;
	L8semprogramacao :=TRUE;
		END_IF
			IF ProducaoProgramada_L8_T2 > 0 AND HabContL8_2T = TRUE THEN 
				L8semprogramacao :=FALSE;
				END_IF
				
IF ProducaoProgramada_L8_T3 = 0 AND HabContL8_3T = TRUE AND TempParadaL8.Q = TRUE THEN
	Status_L8 := 0;
	L8semprogramacao :=TRUE;
		END_IF
			IF ProducaoProgramada_L8_T3 > 0 AND HabContL8_3T = TRUE THEN 
			L8semprogramacao :=FALSE;
			END_IF
	
IF TempParadaL8.Q = FALSE  THEN
	Status_L8 := 1;
END_IF

	IF refeicao = FALSE AND SETUP = FALSE AND DDS = FALSE AND TempParadaL8.Q = TRUE AND L8semprogramacao = FALSE THEN
	Status_L8 := 2;
	END_IF

IF refeicao = TRUE  AND TempParadaL8.Q = TRUE THEN
Status_L8 := 3;
END_IF

IF DDS = TRUE AND TempParadaL8.Q = TRUE THEN
Status_L8 := 4;
END_IF

//IF SETUP = TRUE THEN
//Status_L8 := 5;
//END_IF
//STATUS DA LINHA 8

END_PROGRAM

// ProdL8
PROGRAM ProdL8
VAR
	//PRODUÇÃO LINHAS ENVASE
	
//=========================	
PULSO_CNT_L8_1T: R_TRIG;
PULSO_CNT_L8_2T: R_TRIG;
PULSO_CNT_L8_3T: R_TRIG;
	CNT_PRD_L8: INT;
	CNT_L8: BOOL;
//=========================	
	Result : RTC_STATUS;
	DATEANDTIME : EXTENDED_DATE_AND_TIME;
	xEnable : BOOL;
//=========================		
	dia: INT;
	mes: INT;
	ano: INT;
	hora: INT;
	minuto: INT;
	segundo: INT;
	
	
	
	HoraInicio1Turno: INT;
	MinInicio1Turno: INT;
	HoraFim1Turno: INT;
	MinFim1Turno: INT;
	HoraInicio2Turno: INT;
	MinInicio2Turno: INT;
	HoraFim2Turno: INT;
	MinFim2Turno: INT;
	HoraInicio3Turno: INT;
	MinInicio3Turno: INT;
	HoraFim3Turno: INT;
	MinFim3Turno: INT;
	EficienciaL8: INT;
	ProducaoProgramada_L8_1T: INT;
	ProducaoProgramada_L8_2T: INT;
	ProducaoProgramada_L8_3T: INT;
	HabContL8_1T: BOOL;
	HabContL8_2T: BOOL;
	HabContL8_3T: BOOL;
	CNT_PRD_L8_1T: INT;
	CNT_PRD_L8_2T: INT;
	CNT_PRD_L8_3T: INT;
	EficienciaL8_1T: REAL;
	EficienciaL8_2T: REAL;
	EficienciaL8_3T: REAL;
	
	MinDispL8_1T: REAL;
	EficL8_1T_realtime: REAL;
	ProdL8_1T_realtime: REAL;
	MinDispL8_2T: REAL;
	ProdL8_2T_realtime: REAL;
	EficL8_2T_realtime: REAL;
	MinDispL8_3T: REAL;
	ProdL8_3T_realtime: REAL;
	EficL8_3T_realtime: REAL;
END_VAR


//LÓGICA PARA ANÁLISES DE PRODUTIVADADE DA L8 DE CARTUCHOS
	dia := BYTE_TO_INT (DATEANDTIME.byDayOfMonth);
	mes := BYTE_TO_INT (DATEANDTIME.byMonth);
	ano := WORD_TO_INT (DATEANDTIME.wYear);
	hora := BYTE_TO_INT (DATEANDTIME.byHours);
	minuto := BYTE_TO_INT (DATEANDTIME.byMinutes);
	segundo := BYTE_TO_INT (DATEANDTIME.bySeconds);
	
	
	HoraInicio1Turno := 5;
	MinInicio1Turno := 20;
	HoraFim1Turno := 15;
	MinFim1Turno := 8;
	HoraInicio2Turno := 15;
	MinInicio2Turno := 09;
	HoraFim2Turno := 24;
	MinFim2Turno := 32;
	
	xEnable := TRUE;
//=====================1º TURNO ========================
	
	//10 minutos - Reunião / DSS / Treinamento
	//20 minutosPartida de linha / Parada de Linha
	//15 minutosRefeições (Café / Almoço / Janta)
	//60 minutosRefeições (Café / Almoço / Janta)
	//10 minutosPartida de linha / Parada de Linha
	MinDispL8_1T := (((INT_TO_REAL (HoraFim1Turno) - INT_TO_REAL(HoraInicio1Turno) )*60)-
		INT_TO_REAL(MinInicio1Turno)+INT_TO_REAL(MinFim1Turno)-10-20-15-60-10);
		
	IF hora > 5 AND hora < 7 THEN

		ProdL8_1T_realtime := (INT_TO_REAL(ProducaoProgramada_L8_1T) / (MinDispL8_1T)) * ((
		(INT_TO_REAL(hora)-INT_TO_REAL(HoraInicio1Turno))*60)-INT_TO_REAL(MinInicio1Turno) + INT_TO_REAL(minuto)-10-20);
	
		EficL8_1T_realtime := ( INT_TO_REAL(CNT_PRD_L8_1T) / ProdL8_1T_realtime ) * 100;
		END_IF
		
			IF hora > 7 AND hora < 11 THEN

		ProdL8_1T_realtime := (INT_TO_REAL(ProducaoProgramada_L8_1T) / (MinDispL8_1T)) * ((
		(INT_TO_REAL(hora)-INT_TO_REAL(HoraInicio1Turno))*60)-INT_TO_REAL(MinInicio1Turno) + INT_TO_REAL(minuto)-10-20-15);
	
		EficL8_1T_realtime := ( INT_TO_REAL(CNT_PRD_L8_1T) / ProdL8_1T_realtime ) * 100;
		END_IF
		
				IF hora > 12 AND hora < 15 AND minuto < 9 THEN

		ProdL8_1T_realtime := (INT_TO_REAL(ProducaoProgramada_L8_1T) / (MinDispL8_1T)) * ((
		(INT_TO_REAL(hora)-INT_TO_REAL(HoraInicio1Turno))*60)-INT_TO_REAL(MinInicio1Turno) + INT_TO_REAL(minuto)-10-20-15-60-10);
	
		EficL8_1T_realtime := ( INT_TO_REAL(CNT_PRD_L8_1T) / ProdL8_1T_realtime ) * 100;
		END_IF
//HABILITA RTC==========================
	IF xEnable = TRUE THEN
	Result := GetDateAndTime(DATEANDTIME);
	END_IF
//HABILITA RTC==========================

//==============Habilita contadores 1º turno ================
IF (hora = HoraInicio1Turno AND minuto = MinInicio1Turno)  THEN
HabContL8_1T := TRUE;
HabContL8_3T := FALSE;
END_IF 


//==============Contador e Eficiencia L8 1 TURNO de cartuchos==========
IF HabContL8_1T = TRUE THEN 
PULSO_CNT_L8_1T(CLK:=CNT_L8);	
		IF PULSO_CNT_L8_1T.Q = TRUE THEN
		CNT_PRD_L8_1T := CNT_PRD_L8_1T+1;	
		END_IF
END_IF
EficienciaL8_1T := (INT_TO_REAL(CNT_PRD_L8_1T) / INT_TO_REAL(ProducaoProgramada_L8_1T) ) * 100;

//=====================1º TURNO ========================

//=====================2º TURNO ========================

	//10 minutos - Reunião / DSS / Treinamento
	//20 minutosPartida de linha / Parada de Linha
	//15 minutosRefeições (Café / Almoço / Janta)
	//60 minutosRefeições (Café / Almoço / Janta)
	//10 minutosPartida de linha / Parada de Linha
	IF hora = 0 THEN 
		hora := 24;
	END_IF
	
		MinDispL8_2T := (((INT_TO_REAL (HoraFim2Turno) - INT_TO_REAL(HoraInicio2Turno) )*60)-
		INT_TO_REAL(MinInicio2Turno)+INT_TO_REAL(MinFim2Turno)-10-20-15-60-10);
		
	IF (hora > 15 AND minuto > 8) AND hora < 17 THEN

		ProdL8_2T_realtime := (INT_TO_REAL(ProducaoProgramada_L8_2T) / (MinDispL8_2T)) * ((
		(INT_TO_REAL(hora)-INT_TO_REAL(HoraInicio2Turno))*60)-INT_TO_REAL(MinInicio2Turno) + INT_TO_REAL(minuto)-10-20);
	
		EficL8_2T_realtime := ( INT_TO_REAL(CNT_PRD_L8_2T) / ProdL8_2T_realtime ) * 100;
		END_IF
		
			IF hora > 17 AND hora < 20 THEN

		ProdL8_2T_realtime := (INT_TO_REAL(ProducaoProgramada_L8_2T) / (MinDispL8_2T)) * ((
		(INT_TO_REAL(hora)-INT_TO_REAL(HoraInicio2Turno))*60)-INT_TO_REAL(MinInicio2Turno) + INT_TO_REAL(minuto)-10-20-15);
	
		EficL8_2T_realtime := ( INT_TO_REAL(CNT_PRD_L8_2T) / ProdL8_2T_realtime ) * 100;
		END_IF
		
				IF hora > 20 AND hora < 24 THEN

		ProdL8_2T_realtime := (INT_TO_REAL(ProducaoProgramada_L8_2T) / (MinDispL8_2T)) * ((
		(INT_TO_REAL(hora)-INT_TO_REAL(HoraInicio2Turno))*60)-INT_TO_REAL(MinInicio2Turno) + INT_TO_REAL(minuto)-10-20-15-60-10);
	
		EficL8_2T_realtime := ( INT_TO_REAL(CNT_PRD_L8_2T) / ProdL8_2T_realtime ) * 100;
		END_IF
//==============Contador e Eficiencia L8 2 TURNO de cartuchos==========
//==============Habilita contadores 2º turno ================
IF (hora = HoraInicio2Turno AND minuto = MinInicio2Turno)  THEN
HabContL8_2T := TRUE;
HabContL8_1T := FALSE;
END_IF 
IF HabContL8_2T = TRUE THEN 
PULSO_CNT_L8_2T(CLK:=CNT_L8);	
		IF PULSO_CNT_L8_2T.Q = TRUE THEN
		CNT_PRD_L8_2T := CNT_PRD_L8_2T+1;	
		END_IF
END_IF
EficienciaL8_2T := (INT_TO_REAL (CNT_PRD_L8_2T) / INT_TO_REAL (ProducaoProgramada_L8_2T)  ) * 100;

//=====================2º TURNO ========================

//=====================3º TURNO ========================
//==============Contador e Eficiencia L8 3 TURNO de cartuchos==========

//==============Habilita contadores 3º turno ================
//10 minutos - Reunião / DSS / Treinamento
	//20 minutosPartida de linha / Parada de Linha
	//15 minutosRefeições (Café / Almoço / Janta)
	//60 minutosRefeições (Café / Almoço / Janta)
	//10 minutosPartida de linha / Parada de Linha
	IF hora = 0 THEN 
		hora := 24;
	END_IF
	
		MinDispL8_3T := (((INT_TO_REAL (HoraFim3Turno) - INT_TO_REAL(HoraInicio3Turno) )*60)-
		INT_TO_REAL(MinInicio3Turno)+INT_TO_REAL(MinFim3Turno)-10-20-15-60-10);
		
	IF ((hora > 0 OR hora = 24) AND minuto > 32) AND hora < 02 THEN

		ProdL8_3T_realtime := (INT_TO_REAL(ProducaoProgramada_L8_3T) / (MinDispL8_3T)) * ((
		(INT_TO_REAL(hora)-INT_TO_REAL(HoraInicio3Turno))*60)-INT_TO_REAL(MinInicio3Turno) + INT_TO_REAL(minuto)-10-20);
	
		EficL8_3T_realtime := ( INT_TO_REAL(CNT_PRD_L8_3T) / ProdL8_3T_realtime ) * 100;
		END_IF
		
			IF hora > 17 AND hora < 20 THEN

		ProdL8_3T_realtime := (INT_TO_REAL(ProducaoProgramada_L8_3T) / (MinDispL8_3T)) * ((
		(INT_TO_REAL(hora)-INT_TO_REAL(HoraInicio3Turno))*60)-INT_TO_REAL(MinInicio3Turno) + INT_TO_REAL(minuto)-10-20-15);
	
		EficL8_3T_realtime := ( INT_TO_REAL(CNT_PRD_L8_3T) / ProdL8_3T_realtime ) * 100;
		END_IF
		
				IF hora > 20 AND hora < 24 THEN

		ProdL8_3T_realtime := (INT_TO_REAL(ProducaoProgramada_L8_3T) / (MinDispL8_3T)) * ((
		(INT_TO_REAL(hora)-INT_TO_REAL(HoraInicio3Turno))*60)-INT_TO_REAL(MinInicio3Turno) + INT_TO_REAL(minuto)-10-20-15-60-10);
	
		EficL8_3T_realtime := ( INT_TO_REAL(CNT_PRD_L8_3T) / ProdL8_3T_realtime ) * 100;
		END_IF
//==============Contador e Eficiencia L8 3 TURNO de cartuchos==========
//==============Habilita contadores 3º turno ================
IF (hora = HoraInicio3Turno AND minuto = MinInicio3Turno)  THEN
HabContL8_3T := TRUE;
HabContL8_2T := FALSE;
END_IF 
IF HabContL8_3T = TRUE THEN 
PULSO_CNT_L8_3T(CLK:=CNT_L8);	
		IF PULSO_CNT_L8_3T.Q = TRUE THEN
		CNT_PRD_L8_3T := CNT_PRD_L8_3T+1;	
		END_IF
END_IF
EficienciaL8_3T := (INT_TO_REAL (CNT_PRD_L8_3T) / INT_TO_REAL (ProducaoProgramada_L8_3T)  ) * 100;


IF (hora = HoraInicio3Turno AND minuto = MinInicio3Turno)  THEN
HabContL8_3T := TRUE;
HabContL8_2T := FALSE;
END_IF 
IF HabContL8_3T = TRUE THEN 
PULSO_CNT_L8_3T(CLK:=CNT_L8);	
		IF PULSO_CNT_L8_3T.Q = TRUE THEN
		CNT_PRD_L8_3T := CNT_PRD_L8_3T+1;	
		END_IF
END_IF
EficienciaL8_3T := (INT_TO_REAL (CNT_PRD_L8_3T) / INT_TO_REAL(ProducaoProgramada_L8_3T)  ) * 100;
//=====================3º TURNO ========================

END_PROGRAM

// Device/Application/ProdL9
PROGRAM ProdL9
VAR
	//PRODUÇÃO LINHAS ENVASE
	
//=========================	
PULSO_CNT_L9_1T: R_TRIG;
PULSO_CNT_L9_2T: R_TRIG;
PULSO_CNT_L9_3T: R_TRIG;
	CNT_PRD_L9: INT;
	//CNT_L9: BOOL;
//=========================	
	Result : RTC_STATUS;
	DATEANDTIME : EXTENDED_DATE_AND_TIME;
	xEnable : BOOL;
//=========================		
	dia: INT;
	mes: INT;
	ano: INT;
	hora: INT;
	minuto: INT;
	segundo: INT;
	
	
	
	//HoraInicio1Turno: INT;
	//MinInicio1Turno: INT;
	HoraFim1Turno: INT;
	MinFim1Turno: INT;
	//HoraInicio2Turno: INT;
	//MinInicio2Turno: INT;
	HoraFim2Turno: INT;
	MinFim2Turno: INT;
	//HoraInicio3Turno: INT;
	//MinInicio3Turno: INT;
	HoraFim3Turno: INT;
	MinFim3Turno: INT;
	EficienciaL9: INT;
	
	
	HabContL9_1T: BOOL;
	HabContL9_2T: BOOL;
	HabContL9_3T: BOOL;
	
	CNT_PRD_L9_2T: INT;
	CNT_PRD_L9_3T: INT;
	EficienciaL9_1T: REAL;
	EficienciaL9_2T: REAL;
	EficienciaL9_3T: REAL;
	
	MinDispL9_1T: REAL;
	
	ProdL9_1T_realtime: REAL;
	MinDispL9_2T: REAL;
	ProdL9_2T_realtime: REAL;
	EficL9_2T_realtime: REAL;
	MinDispL9_3T: REAL;
	ProdL9_3T_realtime: REAL;
	EficL9_3T_realtime: REAL;
	
	//TMR_SIMUL_CNT1: TON;
	//LIBERA_TMR_SIMUL: BOOL;
	EficL9_2T_projetada: REAL;
	//TMR_SIMUL_CNT2: TON;
	//LIBERA_TMR_SIMUL9T: BOOL;
	//TMR_SIMUL_CNT3: TON;
	//LIBERA_TMR_SIMUL3T: BOOL;
	EficL9_3T_projetada: REAL;
//	EficL9_1T_realtime: REAL;
	HabTemParadaL9: BOOL;
	TempParadaL9: Ton;
	horaParadaL9: INT;
	MinParadaL9: INT;
	RegistraHora: BOOL;
	Borda_des_RegistraHora: F_TRIG;
	HoraRetornoParadaL9: INT;
	MinRetornoParadaL9: INT;
	TempoParadaL9L9: INT;
	TotalMinParado: TON;
	HabTotalMinParado: BOOL;
	//TempoProduzindoL9: REAL;
	//MinDispTurnoAtual: REAL;

	refeicao: BOOL;
	DDS: BOOL;
	SETUP: BOOL;
	L9semprogramacao: BOOL;
END_VAR


//LÓGICA PARA ANÁLISES DE PRODUTIVADADE DA L9 DE CARTUCHOS
	dia := BYTE_TO_INT (DATEANDTIME.byDayOfMonth);
	mes := BYTE_TO_INT (DATEANDTIME.byMonth);
	ano := WORD_TO_INT (DATEANDTIME.wYear);
	hora := BYTE_TO_INT (DATEANDTIME.byHours);
	minuto := BYTE_TO_INT (DATEANDTIME.byMinutes);
	segundo := BYTE_TO_INT (DATEANDTIME.bySeconds);
	xEnable := TRUE;
	
	//HABILITA RTC==========================
	IF xEnable = TRUE THEN
	Result := GetDateAndTime(DATEANDTIME);
	END_IF
//HABILITA RTC==========================

//=====================1º TURNO ========================
	
		//HoraInicio1Turno: INT;
	
	HoraFim1Turno:= HoraInicio2Turno;
	MinFim1Turno:= MinInicio2Turno;
	HoraFim2Turno:= HoraInicio3Turno;
	MinFim2Turno:= MinInicio3Turno;
	
	//10 minutos - Reunião / DSS / Treinamento
	//20 minutosPartida de linha / Parada de Linha xxxxxxxxxx
	//15 minutosRefeições (Café / Almoço / Janta)xxxxxxxxxxxx
	//60 minutosRefeições (Café / Almoço / Janta)
	//10 minutosPartida de linha / Parada de Linha xxxxxxxxxxxxxx
			
	MinDispL9_1T := (((INT_TO_REAL (HoraFim1Turno) - INT_TO_REAL(HoraInicio1Turno) )*60)-
		INT_TO_REAL(MinInicio1Turno)+INT_TO_REAL(MinFim1Turno)-60-10);
		
			IF TempoProduzindoL9 < 1 THEN
			TempoProduzindoL9 :=0;
		END_IF
	
		//LÓGICA PARA VERIFICAR SE EXISTE ATRASO DE PRODUÇÃO NO INSTANTE ATUAL
		
	
					
	IF  CXS_ATRASOL9 >= 0 AND HabContL9_1T = TRUE THEN 
	CXS_ATRASOL9:= REAL_TO_INT(ProdL9_1T_realtime)-CNT_PRD_L9_1T;
	END_IF
	IF  CXS_ATRASOL9 >= 0 AND HabContL9_2T = TRUE THEN 
	CXS_ATRASOL9:= REAL_TO_INT(ProdL9_2T_realtime)-CNT_PRD_L9_1T;
	END_IF
	IF  CXS_ATRASOL9 >= 0 AND HabContL9_3T = TRUE THEN 
	CXS_ATRASOL9:=REAL_TO_INT(ProdL9_2T_realtime)-CNT_PRD_L9_1T;
	END_IF
		IF  CXS_ATRASOL9  < 0 THEN 
		CXS_ATRASOL9:= 0;
		END_IF
	
	
	//LÓGICA PARA VERIFICAR SE EXISTE ATRASO DE PRODUÇÃO NO INSTANTE ATUAL
		
		//LÓGICA PARA CONTAR TEMPO DE PARADA
		TempParadaL9(IN:=HabTemParadaL9 ,PT:= T#30S);
		IF TempParadaL9.Q   THEN
		TotalMinParado(IN:=HabTotalMinParado ,PT:= T#1M);
		IF TotalMinParado.Q = TRUE THEN
			TempoParadaL9 := TempoParadaL9+1;
			HabTotalMinParado := FALSE;
			ELSE
				HabTotalMinParado := TRUE;
			END_IF
		END_IF
		
		IF PULSO_CNT_L9_1T.Q = FALSE AND PULSO_CNT_L9_2T.Q = FALSE AND PULSO_CNT_L9_3T.Q = FALSE  THEN
		HabTemParadaL9 := TRUE;
		
		ELSE 	
		HabTemParadaL9 := FALSE;
		END_IF
		//LÓGICA PARA CONTAR TEMPO DE PARADA
//==============Habilita contadores 1º turno ================
IF (hora = HoraInicio1Turno AND minuto = MinInicio1Turno)  THEN
HabContL9_1T := TRUE;
HabContL9_3T := FALSE;
HabContL9_2T := FALSE;
CNT_PRD_L9_3T := 0;
CNT_PRD_L9_2T := 0;
CNT_PRD_L9_1T := 0;
TempoProduzindoL9 :=0;
EficL9_1T_projetada:=0;
EficL9_1T_realtime :=0;
ProdL9_1T_realtime :=0;
TempoParadaL9 :=0;
CXS_ATRASOL9:=0;
END_IF 


//==============Contador e Eficiencia L9 1 TURNO de cartuchos==========
IF HabContL9_1T = TRUE THEN 
PULSO_CNT_L9_1T(CLK:=CNT_L9);
//TMR_SIMUL_CNT1(IN:=LIBERA_TMR_SIMUL ,PT:=T#9S);	
		IF PULSO_CNT_L9_1T.Q = TRUE THEN
		CNT_PRD_L9_1T := CNT_PRD_L9_1T+1;
		//LIBERA_TMR_SIMUL := FALSE;
		RegistraHora := FALSE;
		MinDispTurnoAtual := MinDispL9_1T;
//ELSE 	
	//LIBERA_TMR_SIMUL:= TRUE;
		END_IF
		
			IF hora > 5 AND hora < 11 THEN

		ProdL9_1T_realtime := (INT_TO_REAL(ProducaoProgramada_L9_1T) / (MinDispL9_1T)) * ((
		(INT_TO_REAL(hora)-INT_TO_REAL(HoraInicio1Turno))*60)-INT_TO_REAL(MinInicio1Turno) + INT_TO_REAL(minuto));
		
		TempoProduzindoL9 :=  ((hora-HoraInicio1Turno)*60)-MinInicio1Turno+ minuto-TempoParadaL9;
		
		EficL9_1T_realtime := ( INT_TO_REAL(CNT_PRD_L9_1T) / ProdL9_1T_realtime ) * 100 * (EficL9_1T_projetada/100);
		EficL9_1T_projetada := (ProdL9_1T_realtime / ProducaoProgramada_L9_1T) * 100;
		END_IF
		
			IF hora > 11 AND hora < 15 THEN

		ProdL9_1T_realtime := (INT_TO_REAL(ProducaoProgramada_L9_1T) / (MinDispL9_1T)) * ((
		(INT_TO_REAL(hora)-INT_TO_REAL(HoraInicio1Turno))*60)-INT_TO_REAL(MinInicio1Turno) + INT_TO_REAL(minuto)-10-60);
		
		TempoProduzindoL9 :=  ((hora-HoraInicio1Turno)*60)-MinInicio1Turno+ minuto-TempoParadaL9;
		
		EficL9_1T_realtime := ( INT_TO_REAL(CNT_PRD_L9_1T) / ProdL9_1T_realtime ) * 100 * (EficL9_1T_projetada/100);
		EficL9_1T_projetada := (ProdL9_1T_realtime / ProducaoProgramada_L9_1T) * 100;
		END_IF
	
END_IF
EficienciaL9_1T := (INT_TO_REAL(CNT_PRD_L9_1T) / INT_TO_REAL(ProducaoProgramada_L9_1T) ) * 100;


//=====================1º TURNO ========================

//=====================2º TURNO ========================

	//10 minutos - Reunião / DSS / Treinamento
	//20 minutosPartida de linha / Parada de Linha
	//15 minutosRefeições (Café / Almoço / Janta)
	//60 minutosRefeições (Café / Almoço / Janta)
	//10 minutosPartida de linha / Parada de Linha
	IF hora = 0 THEN 
		hora := 24;
	END_IF
	
		MinDispL9_2T := (((INT_TO_REAL (HoraFim2Turno) - INT_TO_REAL(HoraInicio2Turno) )*60)-
		INT_TO_REAL(MinInicio2Turno)+INT_TO_REAL(MinFim2Turno)-60-10);
	
//==============Contador e Eficiencia L9 2 TURNO de cartuchos==========
//==============Habilita contadores 2º turno ================
IF (hora = HoraInicio2Turno AND minuto = MinInicio2Turno)  THEN
HabContL9_2T := TRUE;
HabContL9_1T := FALSE;
CNT_PRD_L9_3T := 0;
CNT_PRD_L9_2T := 0;
CNT_PRD_L9_1T := 0;
TempoParadaL9 :=0;
TempoProduzindoL9 :=0;
EficL9_1T_projetada:=0;
EficL9_1T_realtime :=0;
ProdL9_1T_realtime :=0;
TempoParadaL9 :=0;
CXS_ATRASOL9:=0;
END_IF 
IF HabContL9_2T = TRUE THEN 
PULSO_CNT_L9_2T(CLK:=CNT_L9);
//TMR_SIMUL_CNT2(IN:=LIBERA_TMR_SIMUL9T ,PT:=T#7S);
		IF PULSO_CNT_L9_2T.Q = TRUE  THEN
		CNT_PRD_L9_2T := CNT_PRD_L9_2T+1;
		//LIBERA_TMR_SIMUL9T := FALSE;
		MinDispTurnoAtual := MinDispL9_2T;
//ELSE 	
	//LIBERA_TMR_SIMUL9T:= TRUE;	
		END_IF
		CNT_PRD_L9_1T := CNT_PRD_L9_2T ;
		EficL9_1T_projetada:=EficL9_2T_projetada;
		EficL9_1T_realtime :=EficL9_2T_realtime;
		ProdL9_1T_realtime :=ProdL9_1T_realtime;
		
			IF hora > 13 AND hora < 19 THEN

		ProdL9_2T_realtime := (INT_TO_REAL(ProducaoProgramada_L9_T2) / (MinDispL9_2T)) * ((
		(INT_TO_REAL(hora)-INT_TO_REAL(HoraInicio2Turno))*60)-INT_TO_REAL(MinInicio2Turno) + INT_TO_REAL(minuto));
		
		TempoProduzindoL9 :=  ((hora-HoraInicio2Turno)*60)-MinInicio2Turno+ minuto-TempoParadaL9;
		
		EficL9_2T_realtime := ( INT_TO_REAL(CNT_PRD_L9_2T) / ProdL9_2T_realtime ) * 100 * (EficL9_2T_projetada/100);
		EficL9_2T_projetada := (ProdL9_2T_realtime / ProducaoProgramada_L9_T2) * 100;
		END_IF
		IF hora > 19 AND hora < 23 THEN

		ProdL9_2T_realtime := (INT_TO_REAL(ProducaoProgramada_L9_T2) / (MinDispL9_2T)) * ((
		(INT_TO_REAL(hora)-INT_TO_REAL(HoraInicio2Turno))*60)-INT_TO_REAL(MinInicio2Turno) + INT_TO_REAL(minuto)-10-60);
		
		TempoProduzindoL9 :=  ((hora-HoraInicio2Turno)*60)-MinInicio2Turno+ minuto-TempoParadaL9;
		
		EficL9_2T_realtime := ( INT_TO_REAL(CNT_PRD_L9_2T) / ProdL9_2T_realtime ) * 100 * (EficL9_2T_projetada/100);
		EficL9_2T_projetada := (ProdL9_2T_realtime / ProducaoProgramada_L9_T2) * 100;
		END_IF
END_IF
EficienciaL9_2T := (INT_TO_REAL (CNT_PRD_L9_2T) / INT_TO_REAL (ProducaoProgramada_L9_T2)  ) * 100;

//=====================2º TURNO ========================

//=====================3º TURNO ========================
//==============Contador e Eficiencia L9 3 TURNO de cartuchos==========

//==============Habilita contadores 3º turno ================
//10 minutos - Reunião / DSS / Treinamento
	//20 minutosPartida de linha / Parada de Linha
	//15 minutosRefeições (Café / Almoço / Janta)
	//60 minutosRefeições (Café / Almoço / Janta)
	//10 minutosPartida de linha / Parada de Linha
	IF hora = 0 THEN 
		hora := 24;
	END_IF
	
		MinDispL9_3T := (((INT_TO_REAL (HoraFim3Turno) - INT_TO_REAL(HoraInicio3Turno) )*60)-
		INT_TO_REAL(MinInicio3Turno)+INT_TO_REAL(MinFim3Turno)-60-10);
		
	
//==============Contador e Eficiencia L9 3 TURNO de cartuchos==========
//==============Habilita contadores 3º turno ================
IF (hora = HoraInicio3Turno AND minuto = MinInicio3Turno)  THEN
HabContL9_3T := TRUE;
HabContL9_2T := FALSE;
HabContL9_1T := FALSE;
CNT_PRD_L9_3T := 0;
CNT_PRD_L9_2T := 0;
CNT_PRD_L9_1T := 0;
TempoParadaL9 :=0;
TempoProduzindoL9 :=0;
EficL9_1T_projetada:=0;
EficL9_1T_realtime :=0;
ProdL9_1T_realtime :=0;
TempoParadaL9 :=0;
CXS_ATRASOL9:=0;
END_IF 

IF HabContL9_3T = TRUE THEN 
PULSO_CNT_L9_3T(CLK:=CNT_L9);	
		IF PULSO_CNT_L9_3T.Q = TRUE THEN
		CNT_PRD_L9_3T := CNT_PRD_L9_3T+1;	
			CNT_PRD_L9_1T := CNT_PRD_L9_3T ;
		EficL9_1T_projetada:=EficL9_3T_projetada;
		EficL9_1T_realtime :=EficL9_3T_realtime;
		ProdL9_1T_realtime :=ProdL9_3T_realtime;
		END_IF
		IF hora > 21 AND hora <= 24 THEN

		ProdL9_3T_realtime := (INT_TO_REAL(ProducaoProgramada_L9_T3) / (MinDispL9_3T)) * ((
		(INT_TO_REAL(hora)-INT_TO_REAL(HoraInicio3Turno))*60)-INT_TO_REAL(MinInicio3Turno) + INT_TO_REAL(minuto));
		
		TempoProduzindoL9 :=  ((hora-HoraInicio3Turno)*60)-MinInicio3Turno+ minuto-TempoParadaL9;
	
		EficL9_3T_realtime := ( INT_TO_REAL(CNT_PRD_L9_3T) / ProdL9_3T_realtime ) * 100 *(EficL9_3T_projetada/100) ;
		EficL9_3T_projetada := (ProdL9_3T_realtime / ProducaoProgramada_L9_T3) * 100;
		END_IF
		IF ((hora > 0 ) AND minuto > 30) AND hora < 2 THEN

		ProdL9_3T_realtime := (INT_TO_REAL(ProducaoProgramada_L9_T3) / (MinDispL9_3T)) * ((
		(INT_TO_REAL(hora)-INT_TO_REAL(HoraInicio3Turno))*60)-INT_TO_REAL(MinInicio3Turno) + INT_TO_REAL(minuto)-10-60);
		
		TempoProduzindoL9 :=  ((hora-HoraInicio3Turno)*60)-MinInicio3Turno+ minuto-TempoParadaL9;
	
		EficL9_3T_realtime := ( INT_TO_REAL(CNT_PRD_L9_3T) / ProdL9_3T_realtime ) * 100 *(EficL9_3T_projetada/100) ;
		EficL9_3T_projetada := (ProdL9_3T_realtime / ProducaoProgramada_L9_T3) * 100;
		END_IF
END_IF


EficienciaL9_3T := (INT_TO_REAL (CNT_PRD_L9_3T) / INT_TO_REAL (ProducaoProgramada_L9_T3)  ) * 100;


IF (hora = HoraInicio3Turno AND minuto = MinInicio3Turno)  THEN
HabContL9_3T := TRUE;
HabContL9_2T := FALSE;
END_IF 

IF HabContL9_3T = TRUE THEN 
PULSO_CNT_L9_3T(CLK:=CNT_L9);
//TMR_SIMUL_CNT3(IN:=LIBERA_TMR_SIMUL3T ,PT:=T#8S);
		IF PULSO_CNT_L9_3T.Q = TRUE  THEN
		CNT_PRD_L9_3T := CNT_PRD_L9_3T+1;
		//LIBERA_TMR_SIMUL3T := FALSE;
		MinDispTurnoAtual := MinDispL9_3T;
//ELSE 	
	//LIBERA_TMR_SIMUL3T:= TRUE;	
		END_IF
		END_IF
	
	
EficienciaL9_3T := (INT_TO_REAL (CNT_PRD_L9_3T) / INT_TO_REAL(ProducaoProgramada_L9_T3)  ) * 100;
//=====================3º TURNO ========================

IF (hora = 11 AND minuto = 0) OR (hora = 19 AND minuto = 0) OR (hora = 1 AND minuto = 30)  THEN
	refeicao := TRUE;
	END_IF
	IF (hora = 11 AND minuto = 40) OR  (hora = 20 AND minuto = 0)  OR  (hora = 2 AND minuto = 30)  THEN
	refeicao := FALSE;
	END_IF 
	
	IF (hora = 6 AND minuto = 0) OR (hora = 20 AND minuto = 0) OR (hora = 2 AND minuto = 30)  THEN
	DDS := TRUE;
	END_IF
	IF (hora = 6 AND minuto = 10) OR  (hora = 20 AND minuto = 10)  OR  (hora = 2 AND minuto = 40)  THEN
	DDS := FALSE;
	END_IF 
	IF (hora = 6 AND minuto = 0) OR (hora = 14 AND minuto = 20) OR (hora = 22 AND minuto = 30)  THEN
	SETUP := TRUE;
	END_IF
	IF (hora = 6 AND minuto = 30) OR  (hora = 14 AND minuto = 50)  OR  (hora = 23 AND minuto = 0)  THEN
	SETUP := FALSE;
	END_IF 

//STATUS DA LINHA 9
//STATUS DO EQUIPAMENTO
//0- SEM PROGRAMAÇÃO
//1- PRODUZINDO
//2- PARADA
//3- REFEIÇÃO
//4- DDS
//5- SETUP

IF ProducaoProgramada_L9_1T = 0 AND HabContL9_1T = TRUE AND TempParadaL9.Q = TRUE THEN
	Status_L9 := 0;
	L9semprogramacao :=TRUE;
	END_IF
		IF ProducaoProgramada_L9_1T > 0 AND HabContL9_1T = TRUE THEN 
		L9semprogramacao :=FALSE;
		END_IF
	
IF ProducaoProgramada_L9_T2 = 0 AND HabContL9_2T = TRUE AND TempParadaL9.Q = TRUE THEN
	Status_L9 := 0;
	L9semprogramacao :=TRUE;
		END_IF
			IF ProducaoProgramada_L9_T2 > 0 AND HabContL9_2T = TRUE THEN 
				L9semprogramacao :=FALSE;
				END_IF
				
IF ProducaoProgramada_L9_T3 = 0 AND HabContL9_3T = TRUE AND TempParadaL9.Q = TRUE THEN
	Status_L9 := 0;
	L9semprogramacao :=TRUE;
		END_IF
			IF ProducaoProgramada_L9_T3 > 0 AND HabContL9_3T = TRUE THEN 
			L9semprogramacao :=FALSE;
			END_IF
	
IF TempParadaL9.Q = FALSE  THEN
	Status_L9 := 1;
END_IF

	IF refeicao = FALSE AND SETUP = FALSE AND DDS = FALSE AND TempParadaL9.Q = TRUE AND L9semprogramacao = FALSE THEN
	Status_L9 := 2;
	END_IF

IF refeicao = TRUE AND TempParadaL9.Q = TRUE THEN
Status_L9 := 3;
END_IF

IF DDS = TRUE AND TempParadaL9.Q = TRUE THEN
Status_L9 := 4;
END_IF

//IF SETUP = TRUE THEN
//Status_L9 := 5;
//END_IF
//STATUS DA LINHA 9

END_PROGRAM

// Device/Application/ProdL10
PROGRAM ProdL10
VAR
	//PRODUÇÃO LINHAS ENVASE
	
//=========================	
PULSO_CNT_L10_1T: R_TRIG;
PULSO_CNT_L10_2T: R_TRIG;
PULSO_CNT_L10_3T: R_TRIG;
	CNT_PRD_L10: INT;
	CNT_L10: BOOL;
//=========================	
	Result : RTC_STATUS;
	DATEANDTIME : EXTENDED_DATE_AND_TIME;
	xEnable : BOOL;
//=========================		
	dia: INT;
	mes: INT;
	ano: INT;
	hora: INT;
	minuto: INT;
	segundo: INT;
	
	
	
	HoraInicio1Turno: INT;
	MinInicio1Turno: INT;
	HoraFim1Turno: INT;
	MinFim1Turno: INT;
	HoraInicio2Turno: INT;
	MinInicio2Turno: INT;
	HoraFim2Turno: INT;
	MinFim2Turno: INT;
	HoraInicio3Turno: INT;
	MinInicio3Turno: INT;
	HoraFim3Turno: INT;
	MinFim3Turno: INT;
	EficienciaL10: INT;
	ProducaoProgramada_L10_1T: INT;
	ProducaoProgramada_L10_2T: INT;
	ProducaoProgramada_L10_3T: INT;
	HabContL10_1T: BOOL;
	HabContL10_2T: BOOL;
	HabContL10_3T: BOOL;
	CNT_PRD_L10_1T: INT;
	CNT_PRD_L10_2T: INT;
	CNT_PRD_L10_3T: INT;
	EficienciaL10_1T: REAL;
	EficienciaL10_2T: REAL;
	EficienciaL10_3T: REAL;
	
	MinDispL10_1T: REAL;
	EficL10_1T_realtime: REAL;
	ProdL10_1T_realtime: REAL;
	MinDispL10_2T: REAL;
	ProdL10_2T_realtime: REAL;
	EficL10_2T_realtime: REAL;
	MinDispL10_3T: REAL;
	ProdL10_3T_realtime: REAL;
	EficL10_3T_realtime: REAL;
END_VAR


//LÓGICA PARA ANÁLISES DE PRODUTIVADADE DA L10 DE CARTUCHOS
	dia := BYTE_TO_INT (DATEANDTIME.byDayOfMonth);
	mes := BYTE_TO_INT (DATEANDTIME.byMonth);
	ano := WORD_TO_INT (DATEANDTIME.wYear);
	hora := BYTE_TO_INT (DATEANDTIME.byHours);
	minuto := BYTE_TO_INT (DATEANDTIME.byMinutes);
	segundo := BYTE_TO_INT (DATEANDTIME.bySeconds);
	xEnable := TRUE;
//=====================1º TURNO ========================
	
	//10 minutos - Reunião / DSS / Treinamento
	//20 minutosPartida de linha / Parada de Linha
	//15 minutosRefeições (Café / Almoço / Janta)
	//60 minutosRefeições (Café / Almoço / Janta)
	//10 minutosPartida de linha / Parada de Linha
	MinDispL10_1T := (((INT_TO_REAL (HoraFim1Turno) - INT_TO_REAL(HoraInicio1Turno) )*60)-
		INT_TO_REAL(MinInicio1Turno)+INT_TO_REAL(MinFim1Turno)-10-20-15-60-10);
		
	IF hora > 5 AND hora < 7 THEN

		ProdL10_1T_realtime := (INT_TO_REAL(ProducaoProgramada_L10_1T) / (MinDispL10_1T)) * ((
		(INT_TO_REAL(hora)-INT_TO_REAL(HoraInicio1Turno))*60)-INT_TO_REAL(MinInicio1Turno) + INT_TO_REAL(minuto)-10-20);
	
		EficL10_1T_realtime := ( INT_TO_REAL(CNT_PRD_L10_1T) / ProdL10_1T_realtime ) * 100;
		END_IF
		
			IF hora > 7 AND hora < 11 THEN

		ProdL10_1T_realtime := (INT_TO_REAL(ProducaoProgramada_L10_1T) / (MinDispL10_1T)) * ((
		(INT_TO_REAL(hora)-INT_TO_REAL(HoraInicio1Turno))*60)-INT_TO_REAL(MinInicio1Turno) + INT_TO_REAL(minuto)-10-20-15);
	
		EficL10_1T_realtime := ( INT_TO_REAL(CNT_PRD_L10_1T) / ProdL10_1T_realtime ) * 100;
		END_IF
		
				IF hora > 12 AND hora < 15 AND minuto < 9 THEN

		ProdL10_1T_realtime := (INT_TO_REAL(ProducaoProgramada_L10_1T) / (MinDispL10_1T)) * ((
		(INT_TO_REAL(hora)-INT_TO_REAL(HoraInicio1Turno))*60)-INT_TO_REAL(MinInicio1Turno) + INT_TO_REAL(minuto)-10-20-15-60-10);
	
		EficL10_1T_realtime := ( INT_TO_REAL(CNT_PRD_L10_1T) / ProdL10_1T_realtime ) * 100;
		END_IF
//HABILITA RTC==========================
	IF xEnable = TRUE THEN
	Result := GetDateAndTime(DATEANDTIME);
	END_IF
//HABILITA RTC==========================

//==============Habilita contadores 1º turno ================
IF (hora = HoraInicio1Turno AND minuto = MinInicio1Turno)  THEN
HabContL10_1T := TRUE;
HabContL10_3T := FALSE;
END_IF 


//==============Contador e Eficiencia L10 1 TURNO de cartuchos==========
IF HabContL10_1T = TRUE THEN 
PULSO_CNT_L10_1T(CLK:=CNT_L10);	
		IF PULSO_CNT_L10_1T.Q = TRUE THEN
		CNT_PRD_L10_1T := CNT_PRD_L10_1T+1;	
		END_IF
END_IF
EficienciaL10_1T := (INT_TO_REAL(CNT_PRD_L10_1T) / INT_TO_REAL(ProducaoProgramada_L10_1T) ) * 100;

//=====================1º TURNO ========================

//=====================2º TURNO ========================

	//10 minutos - Reunião / DSS / Treinamento
	//20 minutosPartida de linha / Parada de Linha
	//15 minutosRefeições (Café / Almoço / Janta)
	//60 minutosRefeições (Café / Almoço / Janta)
	//10 minutosPartida de linha / Parada de Linha
	IF hora = 0 THEN 
		hora := 24;
	END_IF
	
		MinDispL10_2T := (((INT_TO_REAL (HoraFim2Turno) - INT_TO_REAL(HoraInicio2Turno) )*60)-
		INT_TO_REAL(MinInicio2Turno)+INT_TO_REAL(MinFim2Turno)-10-20-15-60-10);
		
	IF (hora > 15 AND minuto > 8) AND hora < 17 THEN

		ProdL10_2T_realtime := (INT_TO_REAL(ProducaoProgramada_L10_2T) / (MinDispL10_2T)) * ((
		(INT_TO_REAL(hora)-INT_TO_REAL(HoraInicio2Turno))*60)-INT_TO_REAL(MinInicio2Turno) + INT_TO_REAL(minuto)-10-20);
	
		EficL10_2T_realtime := ( INT_TO_REAL(CNT_PRD_L10_2T) / ProdL10_2T_realtime ) * 100;
		END_IF
		
			IF hora > 17 AND hora < 20 THEN

		ProdL10_2T_realtime := (INT_TO_REAL(ProducaoProgramada_L10_2T) / (MinDispL10_2T)) * ((
		(INT_TO_REAL(hora)-INT_TO_REAL(HoraInicio2Turno))*60)-INT_TO_REAL(MinInicio2Turno) + INT_TO_REAL(minuto)-10-20-15);
	
		EficL10_2T_realtime := ( INT_TO_REAL(CNT_PRD_L10_2T) / ProdL10_2T_realtime ) * 100;
		END_IF
		
				IF hora > 20 AND hora < 24 THEN

		ProdL10_2T_realtime := (INT_TO_REAL(ProducaoProgramada_L10_2T) / (MinDispL10_2T)) * ((
		(INT_TO_REAL(hora)-INT_TO_REAL(HoraInicio2Turno))*60)-INT_TO_REAL(MinInicio2Turno) + INT_TO_REAL(minuto)-10-20-15-60-10);
	
		EficL10_2T_realtime := ( INT_TO_REAL(CNT_PRD_L10_2T) / ProdL10_2T_realtime ) * 100;
		END_IF
//==============Contador e Eficiencia L10 2 TURNO de cartuchos==========
//==============Habilita contadores 2º turno ================
IF (hora = HoraInicio2Turno AND minuto = MinInicio2Turno)  THEN
HabContL10_2T := TRUE;
HabContL10_1T := FALSE;
END_IF 
IF HabContL10_2T = TRUE THEN 
PULSO_CNT_L10_2T(CLK:=CNT_L10);	
		IF PULSO_CNT_L10_2T.Q = TRUE THEN
		CNT_PRD_L10_2T := CNT_PRD_L10_2T+1;	
		END_IF
END_IF
EficienciaL10_2T := (INT_TO_REAL (CNT_PRD_L10_2T) / INT_TO_REAL (ProducaoProgramada_L10_2T)  ) * 100;

//=====================2º TURNO ========================

//=====================3º TURNO ========================
//==============Contador e Eficiencia L10 3 TURNO de cartuchos==========

//==============Habilita contadores 3º turno ================
//10 minutos - Reunião / DSS / Treinamento
	//20 minutosPartida de linha / Parada de Linha
	//15 minutosRefeições (Café / Almoço / Janta)
	//60 minutosRefeições (Café / Almoço / Janta)
	//10 minutosPartida de linha / Parada de Linha
	IF hora = 0 THEN 
		hora := 24;
	END_IF
	
		MinDispL10_3T := (((INT_TO_REAL (HoraFim3Turno) - INT_TO_REAL(HoraInicio3Turno) )*60)-
		INT_TO_REAL(MinInicio3Turno)+INT_TO_REAL(MinFim3Turno)-10-20-15-60-10);
		
	IF ((hora > 0 OR hora = 24) AND minuto > 32) AND hora < 02 THEN

		ProdL10_3T_realtime := (INT_TO_REAL(ProducaoProgramada_L10_3T) / (MinDispL10_3T)) * ((
		(INT_TO_REAL(hora)-INT_TO_REAL(HoraInicio3Turno))*60)-INT_TO_REAL(MinInicio3Turno) + INT_TO_REAL(minuto)-10-20);
	
		EficL10_3T_realtime := ( INT_TO_REAL(CNT_PRD_L10_3T) / ProdL10_3T_realtime ) * 100;
		END_IF
		
			IF hora > 17 AND hora < 20 THEN

		ProdL10_3T_realtime := (INT_TO_REAL(ProducaoProgramada_L10_3T) / (MinDispL10_3T)) * ((
		(INT_TO_REAL(hora)-INT_TO_REAL(HoraInicio3Turno))*60)-INT_TO_REAL(MinInicio3Turno) + INT_TO_REAL(minuto)-10-20-15);
	
		EficL10_3T_realtime := ( INT_TO_REAL(CNT_PRD_L10_3T) / ProdL10_3T_realtime ) * 100;
		END_IF
		
				IF hora > 20 AND hora < 24 THEN

		ProdL10_3T_realtime := (INT_TO_REAL(ProducaoProgramada_L10_3T) / (MinDispL10_3T)) * ((
		(INT_TO_REAL(hora)-INT_TO_REAL(HoraInicio3Turno))*60)-INT_TO_REAL(MinInicio3Turno) + INT_TO_REAL(minuto)-10-20-15-60-10);
	
		EficL10_3T_realtime := ( INT_TO_REAL(CNT_PRD_L10_3T) / ProdL10_3T_realtime ) * 100;
		END_IF
//==============Contador e Eficiencia L10 3 TURNO de cartuchos==========
//==============Habilita contadores 3º turno ================
IF (hora = HoraInicio3Turno AND minuto = MinInicio3Turno)  THEN
HabContL10_3T := TRUE;
HabContL10_2T := FALSE;
END_IF 
IF HabContL10_3T = TRUE THEN 
PULSO_CNT_L10_3T(CLK:=CNT_L10);	
		IF PULSO_CNT_L10_3T.Q = TRUE THEN
		CNT_PRD_L10_3T := CNT_PRD_L10_3T+1;	
		END_IF
END_IF
EficienciaL10_3T := (INT_TO_REAL (CNT_PRD_L10_3T) / INT_TO_REAL (ProducaoProgramada_L10_3T)  ) * 100;


IF (hora = HoraInicio3Turno AND minuto = MinInicio3Turno)  THEN
HabContL10_3T := TRUE;
HabContL10_2T := FALSE;
END_IF 
IF HabContL10_3T = TRUE THEN 
PULSO_CNT_L10_3T(CLK:=CNT_L10);	
		IF PULSO_CNT_L10_3T.Q = TRUE THEN
		CNT_PRD_L10_3T := CNT_PRD_L10_3T+1;	
		END_IF
END_IF
EficienciaL10_3T := (INT_TO_REAL (CNT_PRD_L10_3T) / INT_TO_REAL(ProducaoProgramada_L10_3T)  ) * 100;
//=====================3º TURNO ========================

END_PROGRAM

// Device/Application/ProdAerossol
PROGRAM ProdAerossol
VAR
	//PRODUÇÃO LINHAS ENVASE
	
//=========================	
PULSO_CNT_AER_1T: R_TRIG;
PULSO_CNT_AER_2T: R_TRIG;
PULSO_CNT_AER_3T: R_TRIG;
	CNT_PRD_AER: INT;
	CNT_AER: BOOL;
//=========================	
	Result : RTC_STATUS;
	DATEANDTIME : EXTENDED_DATE_AND_TIME;
	xEnable : BOOL;
//=========================		
	dia: INT;
	mes: INT;
	ano: INT;
	hora: INT;
	minuto: INT;
	segundo: INT;
	
	
	
	HoraInicio1Turno: INT;
	MinInicio1Turno: INT;
	HoraFim1Turno: INT;
	MinFim1Turno: INT;
	HoraInicio2Turno: INT;
	MinInicio2Turno: INT;
	HoraFim2Turno: INT;
	MinFim2Turno: INT;
	HoraInicio3Turno: INT;
	MinInicio3Turno: INT;
	HoraFim3Turno: INT;
	MinFim3Turno: INT;
	EficienciaAER: INT;
	ProducaoProgramada_AER_1T: INT;
	ProducaoProgramada_AER_2T: INT;
	ProducaoProgramada_AER_3T: INT;
	HabContAER_1T: BOOL;
	HabContAER_2T: BOOL;
	HabContAER_3T: BOOL;
	CNT_PRD_AER_1T: INT;
	CNT_PRD_AER_2T: INT;
	CNT_PRD_AER_3T: INT;
	EficienciaAER_1T: REAL;
	EficienciaAER_2T: REAL;
	EficienciaAER_3T: REAL;
	
	MinDispAER_1T: REAL;
	EficAER_1T_realtime: REAL;
	ProdAER_1T_realtime: REAL;
	MinDispAER_2T: REAL;
	ProdAER_2T_realtime: REAL;
	EficAER_2T_realtime: REAL;
	MinDispAER_3T: REAL;
	ProdAER_3T_realtime: REAL;
	EficAER_3T_realtime: REAL;
END_VAR


//LÓGICA PARA ANÁLISES DE PRODUTIVADADE DA AER DE CARTUCHOS
	dia := BYTE_TO_INT (DATEANDTIME.byDayOfMonth);
	mes := BYTE_TO_INT (DATEANDTIME.byMonth);
	ano := WORD_TO_INT (DATEANDTIME.wYear);
	hora := BYTE_TO_INT (DATEANDTIME.byHours);
	minuto := BYTE_TO_INT (DATEANDTIME.byMinutes);
	segundo := BYTE_TO_INT (DATEANDTIME.bySeconds);
	xEnable := TRUE;
//=====================1º TURNO ========================
	
	//10 minutos - Reunião / DSS / Treinamento
	//20 minutosPartida de linha / Parada de Linha
	//15 minutosRefeições (Café / Almoço / Janta)
	//60 minutosRefeições (Café / Almoço / Janta)
	//10 minutosPartida de linha / Parada de Linha
	MinDispAER_1T := (((INT_TO_REAL (HoraFim1Turno) - INT_TO_REAL(HoraInicio1Turno) )*60)-
		INT_TO_REAL(MinInicio1Turno)+INT_TO_REAL(MinFim1Turno)-10-20-15-60-10);
		
	IF hora > 5 AND hora < 7 THEN

		ProdAER_1T_realtime := (INT_TO_REAL(ProducaoProgramada_AER_1T) / (MinDispAER_1T)) * ((
		(INT_TO_REAL(hora)-INT_TO_REAL(HoraInicio1Turno))*60)-INT_TO_REAL(MinInicio1Turno) + INT_TO_REAL(minuto)-10-20);
	
		EficAER_1T_realtime := ( INT_TO_REAL(CNT_PRD_AER_1T) / ProdAER_1T_realtime ) * 100;
		END_IF
		
			IF hora > 7 AND hora < 11 THEN

